Yaskawa INFORM job: A_ROOF_UPPER_0614_2_PAINT_2.JBI

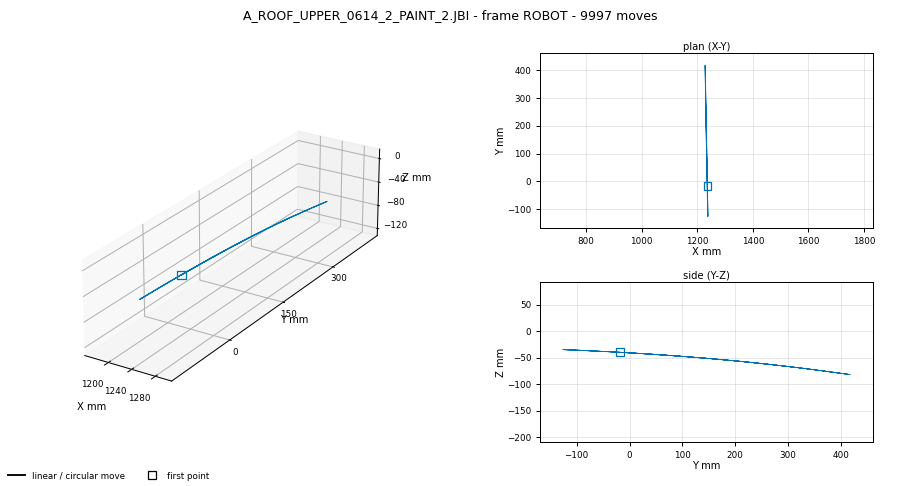
[picture p0: tool path of A_ROOF_UPPER_0614_2_PAINT_2.JBI in frame ROBOT, 9997 of 9997 moves have a stored position in this frame; points joined in program order, loops and branches not executed]
/JOB
//NAME A_ROOF_UPPER_0614_2_PAINT2
//POS
///NPOS 9997,0,0,0,0,0
///TOOL 1
///USER 0
///POSTYPE ROBOT
///RECTAN
///RCONF 1,0,0,0,0,0,0,0,0,0,0,0,0,0,0,0,0,0,0,0,0,0,0,0
C00000=1236.915,-17.452,-39.644,-179.558,5.242,148.773
C00001=1236.910,-17.203,-39.658,-179.555,5.243,148.772
C00002=1236.905,-16.953,-39.672,-179.553,5.243,148.771
C00003=1236.900,-16.704,-39.686,-179.551,5.243,148.771
C00004=1236.895,-16.454,-39.700,-179.548,5.244,148.770
C00005=1236.890,-16.204,-39.714,-179.546,5.243,148.769
C00006=1236.884,-15.955,-39.728,-179.543,5.244,148.769
C00007=1236.880,-15.705,-39.741,-179.541,5.244,148.768
C00008=1236.875,-15.456,-39.756,-179.539,5.244,148.767
C00009=1236.870,-15.206,-39.770,-179.536,5.245,148.767
C00010=1236.864,-14.956,-39.783,-179.534,5.244,148.766
C00011=1236.859,-14.707,-39.798,-179.531,5.245,148.765
C00012=1236.854,-14.457,-39.812,-179.528,5.245,148.764
C00013=1236.849,-14.207,-39.826,-179.526,5.245,148.764
C00014=1236.844,-13.959,-39.839,-179.523,5.245,148.763
C00015=1236.839,-13.709,-39.854,-179.521,5.246,148.762
C00016=1236.834,-13.459,-39.868,-179.519,5.246,148.761
C00017=1236.829,-13.209,-39.882,-179.516,5.246,148.761
C00018=1236.824,-12.960,-39.896,-179.513,5.247,148.760
C00019=1236.819,-12.711,-39.910,-179.511,5.246,148.759
C00020=1236.814,-12.461,-39.925,-179.508,5.247,148.759
C00021=1236.809,-12.211,-39.938,-179.506,5.247,148.758
C00022=1236.803,-11.962,-39.952,-179.504,5.247,148.757
C00023=1236.799,-11.712,-39.966,-179.501,5.248,148.757
C00024=1236.794,-11.463,-39.980,-179.499,5.247,148.756
C00025=1236.789,-11.213,-39.994,-179.496,5.248,148.755
C00026=1236.784,-10.964,-40.008,-179.494,5.248,148.755
C00027=1236.779,-10.714,-40.023,-179.492,5.248,148.754
C00028=1236.774,-10.464,-40.037,-179.488,5.248,148.753
C00029=1236.769,-10.215,-40.051,-179.486,5.249,148.752
C00030=1236.764,-9.965,-40.065,-179.484,5.249,148.752
C00031=1236.758,-9.716,-40.079,-179.481,5.249,148.751
C00032=1236.753,-9.466,-40.094,-179.478,5.250,148.750
C00033=1236.748,-9.217,-40.108,-179.476,5.249,148.749
C00034=1236.743,-8.967,-40.122,-179.474,5.250,148.749
C00035=1236.739,-8.718,-40.137,-179.471,5.250,148.748
C00036=1236.734,-8.468,-40.151,-179.469,5.250,148.747
C00037=1236.728,-8.219,-40.165,-179.466,5.251,148.747
C00038=1236.723,-7.969,-40.180,-179.464,5.251,148.746
C00039=1236.718,-7.720,-40.194,-179.462,5.251,148.745
C00040=1236.713,-7.470,-40.208,-179.459,5.251,148.745
C00041=1236.708,-7.220,-40.222,-179.456,5.252,148.744
C00042=1236.703,-6.970,-40.237,-179.454,5.252,148.743
C00043=1236.698,-6.721,-40.251,-179.451,5.252,148.743
C00044=1236.693,-6.472,-40.265,-179.448,5.252,148.742
C00045=1236.688,-6.223,-40.280,-179.446,5.252,148.741
C00046=1236.683,-5.973,-40.294,-179.444,5.253,148.740
C00047=1236.678,-5.723,-40.308,-179.441,5.253,148.740
C00048=1236.673,-5.474,-40.323,-179.439,5.253,148.739
C00049=1236.668,-5.224,-40.337,-179.436,5.253,148.738
C00050=1236.663,-4.975,-40.351,-179.434,5.254,148.737
C00051=1236.658,-4.725,-40.365,-179.431,5.254,148.737
C00052=1236.653,-4.476,-40.380,-179.429,5.254,148.736
C00053=1236.648,-4.226,-40.394,-179.426,5.255,148.735
C00054=1236.643,-3.976,-40.409,-179.424,5.254,148.735
C00055=1236.638,-3.727,-40.424,-179.421,5.255,148.734
C00056=1236.633,-3.477,-40.438,-179.419,5.255,148.733
C00057=1236.628,-3.228,-40.453,-179.417,5.255,148.733
C00058=1236.623,-2.978,-40.467,-179.414,5.256,148.732
C00059=1236.617,-2.729,-40.481,-179.411,5.256,148.731
C00060=1236.613,-2.479,-40.495,-179.409,5.256,148.731
C00061=1236.608,-2.230,-40.510,-179.407,5.256,148.730
C00062=1236.603,-1.981,-40.525,-179.404,5.257,148.729
C00063=1236.597,-1.731,-40.540,-179.401,5.256,148.728
C00064=1236.592,-1.481,-40.554,-179.399,5.257,148.728
C00065=1236.588,-1.232,-40.569,-179.396,5.257,148.727
C00066=1236.583,-0.982,-40.583,-179.394,5.257,148.726
C00067=1236.578,-0.732,-40.597,-179.391,5.258,148.725
C00068=1236.573,-0.483,-40.612,-179.389,5.258,148.725
C00069=1236.568,-0.233,-40.627,-179.387,5.258,148.724
C00070=1236.562,0.017,-40.641,-179.384,5.258,148.723
C00071=1236.558,0.266,-40.656,-179.381,5.259,148.723
C00072=1236.552,0.515,-40.670,-179.379,5.259,148.722
C00073=1236.547,0.764,-40.685,-179.377,5.259,148.721
C00074=1236.543,1.013,-40.700,-179.374,5.260,148.721
C00075=1236.537,1.263,-40.715,-179.371,5.260,148.720
C00076=1236.532,1.513,-40.729,-179.369,5.260,148.719
C00077=1236.527,1.762,-40.744,-179.367,5.261,148.719
C00078=1236.522,2.012,-40.758,-179.364,5.261,148.718
C00079=1236.518,2.261,-40.773,-179.362,5.261,148.717
C00080=1236.512,2.511,-40.788,-179.359,5.261,148.717
C00081=1236.507,2.761,-40.802,-179.357,5.262,148.716
C00082=1236.502,3.010,-40.817,-179.354,5.262,148.715
C00083=1236.497,3.260,-40.831,-179.352,5.262,148.714
C00084=1236.492,3.529,-40.848,-179.349,5.262,148.714
C00085=1236.486,3.797,-40.863,-179.346,5.263,148.713
C00086=1236.481,4.066,-40.879,-179.343,5.263,148.712
C00087=1236.475,4.335,-40.895,-179.341,5.263,148.711
C00088=1236.471,4.584,-40.910,-179.338,5.263,148.711
C00089=1236.466,4.834,-40.925,-179.335,5.264,148.710
C00090=1236.461,5.083,-40.940,-179.333,5.264,148.709
C00091=1236.456,5.333,-40.955,-179.331,5.264,148.709
C00092=1236.451,5.582,-40.970,-179.328,5.265,148.708
C00093=1236.446,5.832,-40.984,-179.325,5.265,148.707
C00094=1236.441,6.082,-40.999,-179.323,5.265,148.706
C00095=1236.436,6.331,-41.014,-179.321,5.265,148.706
C00096=1236.431,6.580,-41.029,-179.318,5.266,148.705
C00097=1236.425,6.830,-41.044,-179.315,5.266,148.704
C00098=1236.421,7.079,-41.059,-179.313,5.266,148.704
C00099=1236.416,7.329,-41.073,-179.311,5.267,148.703
C00100=1236.410,7.579,-41.088,-179.308,5.267,148.702
C00101=1236.405,7.828,-41.103,-179.306,5.267,148.702
C00102=1236.401,8.077,-41.118,-179.303,5.268,148.701
C00103=1236.395,8.327,-41.133,-179.301,5.268,148.700
C00104=1236.391,8.577,-41.148,-179.298,5.269,148.700
C00105=1236.386,8.826,-41.163,-179.296,5.268,148.699
C00106=1236.381,9.076,-41.178,-179.293,5.269,148.698
C00107=1236.376,9.325,-41.193,-179.291,5.269,148.698
C00108=1236.371,9.575,-41.207,-179.289,5.269,148.697
C00109=1236.366,9.824,-41.223,-179.286,5.270,148.696
C00110=1236.361,10.074,-41.238,-179.283,5.270,148.695
C00111=1236.355,10.324,-41.253,-179.281,5.271,148.695
C00112=1236.351,10.573,-41.268,-179.279,5.271,148.694
C00113=1236.346,10.822,-41.283,-179.276,5.271,148.693
C00114=1236.340,11.072,-41.297,-179.273,5.272,148.693
C00115=1236.336,11.321,-41.312,-179.271,5.271,148.692
C00116=1236.331,11.571,-41.328,-179.268,5.272,148.691
C00117=1236.326,11.821,-41.343,-179.265,5.272,148.690
C00118=1236.320,12.070,-41.358,-179.263,5.273,148.690
C00119=1236.316,12.319,-41.373,-179.261,5.272,148.689
C00120=1236.311,12.569,-41.388,-179.258,5.273,148.688
C00121=1236.305,12.818,-41.403,-179.255,5.273,148.688
C00122=1236.301,13.067,-41.418,-179.253,5.274,148.687
C00123=1236.295,13.317,-41.434,-179.251,5.274,148.686
C00124=1236.291,13.567,-41.448,-179.248,5.274,148.686
C00125=1236.286,13.817,-41.464,-179.245,5.275,148.685
C00126=1236.281,14.066,-41.479,-179.243,5.275,148.684
C00127=1236.276,14.315,-41.494,-179.241,5.275,148.684
C00128=1236.271,14.565,-41.509,-179.238,5.276,148.683
C00129=1236.265,14.814,-41.524,-179.235,5.276,148.682
C00130=1236.261,15.063,-41.539,-179.233,5.276,148.682
C00131=1236.256,15.313,-41.555,-179.231,5.276,148.681
C00132=1236.251,15.562,-41.570,-179.228,5.277,148.680
C00133=1236.246,15.813,-41.585,-179.225,5.278,148.679
C00134=1236.241,16.062,-41.600,-179.223,5.277,148.679
C00135=1236.236,16.311,-41.616,-179.221,5.278,148.678
C00136=1236.231,16.560,-41.631,-179.218,5.278,148.677
C00137=1236.226,16.810,-41.647,-179.215,5.279,148.677
C00138=1236.221,17.059,-41.662,-179.213,5.279,148.676
C00139=1236.216,17.309,-41.677,-179.211,5.279,148.675
C00140=1236.210,17.559,-41.692,-179.208,5.280,148.675
C00141=1236.206,17.808,-41.707,-179.205,5.280,148.674
C00142=1236.201,18.058,-41.723,-179.203,5.280,148.673
C00143=1236.196,18.307,-41.738,-179.201,5.281,148.673
C00144=1236.191,18.556,-41.754,-179.198,5.281,148.672
C00145=1236.186,18.805,-41.769,-179.195,5.282,148.671
C00146=1236.181,19.055,-41.784,-179.193,5.281,148.671
C00147=1236.176,19.305,-41.800,-179.190,5.282,148.670
C00148=1236.171,19.554,-41.815,-179.188,5.283,148.669
C00149=1236.166,19.804,-41.830,-179.185,5.283,148.669
C00150=1236.161,20.053,-41.845,-179.183,5.283,148.668
C00151=1236.156,20.303,-41.861,-179.180,5.283,148.667
C00152=1236.151,20.553,-41.877,-179.178,5.284,148.666
C00153=1236.146,20.802,-41.892,-179.175,5.284,148.666
C00154=1236.141,21.051,-41.907,-179.173,5.284,148.665
C00155=1236.135,21.301,-41.923,-179.170,5.285,148.664
C00156=1236.131,21.550,-41.938,-179.168,5.285,148.664
C00157=1236.126,21.800,-41.954,-179.165,5.286,148.663
C00158=1236.121,22.049,-41.969,-179.163,5.286,148.662
C00159=1236.116,22.298,-41.984,-179.160,5.286,148.662
C00160=1236.111,22.548,-42.000,-179.158,5.287,148.661
C00161=1236.107,22.797,-42.015,-179.155,5.287,148.660
C00162=1236.101,23.047,-42.031,-179.153,5.288,148.660
C00163=1236.096,23.297,-42.047,-179.150,5.288,148.659
C00164=1236.091,23.546,-42.062,-179.148,5.288,148.658
C00165=1236.086,23.795,-42.077,-179.145,5.289,148.658
C00166=1236.081,24.044,-42.094,-179.143,5.289,148.657
C00167=1236.076,24.294,-42.110,-179.140,5.289,148.656
C00168=1236.072,24.543,-42.125,-179.138,5.290,148.656
C00169=1236.066,24.793,-42.140,-179.135,5.290,148.655
C00170=1236.062,25.043,-42.156,-179.132,5.291,148.654
C00171=1236.057,25.292,-42.171,-179.130,5.291,148.654
C00172=1236.052,25.541,-42.187,-179.128,5.291,148.653
C00173=1236.047,25.792,-42.203,-179.125,5.291,148.652
C00174=1236.041,26.041,-42.218,-179.122,5.292,148.652
C00175=1236.037,26.289,-42.234,-179.120,5.293,148.651
C00176=1236.032,26.539,-42.250,-179.118,5.292,148.650
C00177=1236.027,26.789,-42.266,-179.115,5.293,148.649
C00178=1236.022,27.038,-42.281,-179.112,5.293,148.649
C00179=1236.017,27.287,-42.296,-179.110,5.294,148.648
C00180=1236.012,27.538,-42.312,-179.107,5.295,148.647
C00181=1236.007,27.786,-42.328,-179.105,5.294,148.647
C00182=1236.002,28.036,-42.344,-179.102,5.295,148.646
C00183=1235.997,28.286,-42.360,-179.100,5.295,148.645
C00184=1235.992,28.535,-42.375,-179.097,5.296,148.645
C00185=1235.987,28.785,-42.391,-179.095,5.296,148.644
C00186=1235.982,29.034,-42.407,-179.092,5.296,148.643
C00187=1235.977,29.283,-42.423,-179.090,5.297,148.643
C00188=1235.971,29.552,-42.440,-179.087,5.297,148.642
C00189=1235.966,29.821,-42.457,-179.085,5.298,148.641
C00190=1235.961,30.089,-42.474,-179.081,5.298,148.640
C00191=1235.956,30.358,-42.491,-179.079,5.299,148.640
C00192=1235.951,30.607,-42.506,-179.076,5.299,148.639
C00193=1235.946,30.857,-42.522,-179.074,5.299,148.638
C00194=1235.941,31.106,-42.538,-179.071,5.300,148.638
C00195=1235.936,31.356,-42.554,-179.069,5.300,148.637
C00196=1235.931,31.605,-42.570,-179.066,5.301,148.636
C00197=1235.926,31.854,-42.586,-179.063,5.301,148.636
C00198=1235.922,32.104,-42.602,-179.061,5.301,148.635
C00199=1235.916,32.353,-42.617,-179.059,5.302,148.634
C00200=1235.912,32.603,-42.634,-179.056,5.302,148.634
C00201=1235.906,32.852,-42.649,-179.053,5.303,148.633
C00202=1235.901,33.102,-42.665,-179.051,5.303,148.632
C00203=1235.896,33.351,-42.682,-179.049,5.303,148.632
C00204=1235.891,33.600,-42.697,-179.046,5.304,148.631
C00205=1235.886,33.851,-42.713,-179.043,5.304,148.630
C00206=1235.881,34.099,-42.730,-179.041,5.305,148.630
C00207=1235.876,34.349,-42.746,-179.038,5.305,148.629
C00208=1235.871,34.598,-42.762,-179.037,5.305,148.628
C00209=1235.867,34.847,-42.777,-179.034,5.306,148.628
C00210=1235.862,35.097,-42.794,-179.031,5.307,148.627
C00211=1235.857,35.346,-42.809,-179.029,5.307,148.626
C00212=1235.852,35.596,-42.825,-179.026,5.308,148.626
C00213=1235.847,35.845,-42.841,-179.023,5.308,148.625
C00214=1235.842,36.095,-42.857,-179.021,5.308,148.624
C00215=1235.837,36.344,-42.874,-179.019,5.309,148.624
C00216=1235.832,36.594,-42.890,-179.016,5.309,148.623
C00217=1235.827,36.843,-42.906,-179.013,5.310,148.622
C00218=1235.822,37.093,-42.922,-179.011,5.310,148.622
C00219=1235.817,37.342,-42.938,-179.009,5.310,148.621
C00220=1235.813,37.592,-42.954,-179.006,5.311,148.620
C00221=1235.807,37.841,-42.970,-179.003,5.311,148.620
C00222=1235.803,38.091,-42.986,-179.001,5.312,148.619
C00223=1235.798,38.340,-43.003,-178.998,5.312,148.618
C00224=1235.793,38.590,-43.019,-178.995,5.313,148.618
C00225=1235.788,38.838,-43.035,-178.993,5.313,148.617
C00226=1235.783,39.089,-43.051,-178.991,5.313,148.616
C00227=1235.778,39.337,-43.067,-178.988,5.314,148.616
C00228=1235.773,39.587,-43.084,-178.985,5.314,148.615
C00229=1235.767,39.837,-43.100,-178.983,5.315,148.614
C00230=1235.763,40.086,-43.117,-178.980,5.315,148.614
C00231=1235.757,40.335,-43.132,-178.978,5.315,148.613
C00232=1235.753,40.585,-43.149,-178.975,5.316,148.612
C00233=1235.747,40.834,-43.165,-178.973,5.316,148.612
C00234=1235.743,41.084,-43.181,-178.971,5.317,148.611
C00235=1235.738,41.333,-43.197,-178.968,5.318,148.610
C00236=1235.733,41.583,-43.213,-178.965,5.318,148.610
C00237=1235.728,41.831,-43.230,-178.963,5.318,148.609
C00238=1235.724,42.081,-43.246,-178.961,5.319,148.608
C00239=1235.718,42.330,-43.262,-178.958,5.319,148.608
C00240=1235.713,42.580,-43.279,-178.955,5.320,148.607
C00241=1235.708,42.829,-43.296,-178.953,5.320,148.606
C00242=1235.703,43.079,-43.312,-178.950,5.321,148.606
C00243=1235.699,43.329,-43.328,-178.948,5.322,148.605
C00244=1235.694,43.577,-43.345,-178.945,5.321,148.604
C00245=1235.689,43.827,-43.360,-178.943,5.322,148.604
C00246=1235.684,44.076,-43.377,-178.940,5.322,148.603
C00247=1235.678,44.326,-43.394,-178.938,5.323,148.602
C00248=1235.674,44.575,-43.411,-178.935,5.324,148.602
C00249=1235.669,44.825,-43.426,-178.932,5.324,148.601
C00250=1235.664,45.074,-43.443,-178.930,5.325,148.600
C00251=1235.659,45.323,-43.459,-178.928,5.324,148.600
C00252=1235.655,45.573,-43.476,-178.925,5.325,148.599
C00253=1235.648,45.822,-43.492,-178.923,5.326,148.599
C00254=1235.644,46.072,-43.509,-178.920,5.327,148.598
C00255=1235.639,46.321,-43.525,-178.917,5.327,148.597
C00256=1235.634,46.570,-43.542,-178.915,5.328,148.596
C00257=1235.630,46.820,-43.558,-178.912,5.328,148.596
C00258=1235.624,47.070,-43.575,-178.910,5.328,148.595
C00259=1235.619,47.319,-43.591,-178.908,5.329,148.594
C00260=1235.615,47.568,-43.608,-178.905,5.329,148.594
C00261=1235.610,47.817,-43.624,-178.902,5.330,148.593
C00262=1235.605,48.067,-43.642,-178.900,5.330,148.592
C00263=1235.600,48.317,-43.657,-178.897,5.331,148.592
C00264=1235.595,48.566,-43.674,-178.894,5.331,148.591
C00265=1235.590,48.815,-43.690,-178.892,5.331,148.590
C00266=1235.585,49.065,-43.708,-178.890,5.332,148.590
C00267=1235.580,49.314,-43.724,-178.887,5.333,148.589
C00268=1235.575,49.563,-43.741,-178.885,5.333,148.589
C00269=1235.571,49.813,-43.757,-178.882,5.334,148.588
C00270=1235.565,50.062,-43.774,-178.880,5.334,148.587
C00271=1235.561,50.311,-43.791,-178.877,5.335,148.587
C00272=1235.556,50.561,-43.808,-178.874,5.336,148.586
C00273=1235.550,50.811,-43.824,-178.872,5.335,148.585
C00274=1235.546,51.060,-43.840,-178.870,5.336,148.585
C00275=1235.541,51.309,-43.857,-178.867,5.337,148.584
C00276=1235.535,51.559,-43.874,-178.864,5.337,148.583
C00277=1235.531,51.808,-43.891,-178.862,5.338,148.583
C00278=1235.526,52.058,-43.907,-178.859,5.338,148.582
C00279=1235.521,52.307,-43.925,-178.857,5.339,148.582
C00280=1235.516,52.556,-43.941,-178.854,5.340,148.581
C00281=1235.511,52.806,-43.958,-178.852,5.340,148.580
C00282=1235.506,53.055,-43.975,-178.850,5.340,148.580
C00283=1235.501,53.304,-43.991,-178.847,5.341,148.579
C00284=1235.497,53.554,-44.008,-178.844,5.341,148.578
C00285=1235.491,53.803,-44.025,-178.842,5.342,148.577
C00286=1235.487,54.053,-44.042,-178.839,5.342,148.577
C00287=1235.482,54.302,-44.058,-178.836,5.343,148.576
C00288=1235.477,54.552,-44.075,-178.834,5.344,148.575
C00289=1235.473,54.800,-44.093,-178.831,5.344,148.575
C00290=1235.467,55.049,-44.110,-178.829,5.345,148.574
C00291=1235.462,55.299,-44.126,-178.826,5.346,148.574
C00292=1235.457,55.568,-44.145,-178.823,5.346,148.573
C00293=1235.452,55.836,-44.163,-178.821,5.347,148.572
C00294=1235.446,56.105,-44.181,-178.818,5.347,148.571
C00295=1235.441,56.372,-44.199,-178.815,5.348,148.571
C00296=1235.436,56.622,-44.216,-178.813,5.348,148.570
C00297=1235.431,56.872,-44.233,-178.810,5.349,148.569
C00298=1235.427,57.121,-44.250,-178.808,5.349,148.569
C00299=1235.422,57.371,-44.267,-178.806,5.350,148.568
C00300=1235.416,57.620,-44.283,-178.803,5.350,148.568
C00301=1235.411,57.870,-44.301,-178.801,5.351,148.567
C00302=1235.407,58.118,-44.318,-178.798,5.351,148.566
C00303=1235.402,58.368,-44.335,-178.795,5.352,148.566
C00304=1235.397,58.617,-44.352,-178.793,5.352,148.565
C00305=1235.392,58.867,-44.369,-178.790,5.353,148.564
C00306=1235.387,59.116,-44.385,-178.787,5.354,148.564
C00307=1235.382,59.365,-44.403,-178.785,5.354,148.563
C00308=1235.378,59.615,-44.420,-178.782,5.355,148.562
C00309=1235.372,59.864,-44.437,-178.781,5.355,148.562
C00310=1235.367,60.114,-44.454,-178.778,5.356,148.561
C00311=1235.362,60.363,-44.472,-178.775,5.356,148.561
C00312=1235.358,60.612,-44.488,-178.773,5.357,148.560
C00313=1235.353,60.862,-44.506,-178.770,5.357,148.559
C00314=1235.348,61.111,-44.522,-178.767,5.358,148.559
C00315=1235.343,61.360,-44.540,-178.765,5.358,148.558
C00316=1235.338,61.610,-44.557,-178.762,5.359,148.557
C00317=1235.333,61.859,-44.574,-178.759,5.360,148.557
C00318=1235.328,62.108,-44.592,-178.757,5.361,148.556
C00319=1235.324,62.358,-44.608,-178.755,5.361,148.556
C00320=1235.318,62.608,-44.626,-178.752,5.362,148.555
C00321=1235.314,62.857,-44.642,-178.749,5.362,148.554
C00322=1235.309,63.106,-44.660,-178.747,5.363,148.554
C00323=1235.303,63.355,-44.677,-178.745,5.363,148.553
C00324=1235.299,63.604,-44.695,-178.742,5.363,148.552
C00325=1235.294,63.854,-44.712,-178.739,5.364,148.552
C00326=1235.289,64.104,-44.729,-178.737,5.365,148.551
C00327=1235.285,64.353,-44.747,-178.735,5.365,148.550
C00328=1235.279,64.603,-44.764,-178.732,5.366,148.550
C00329=1235.275,64.852,-44.780,-178.729,5.367,148.549
C00330=1235.269,65.100,-44.798,-178.727,5.367,148.548
C00331=1235.264,65.350,-44.815,-178.724,5.368,148.548
C00332=1235.260,65.599,-44.833,-178.722,5.368,148.547
C00333=1235.255,65.849,-44.850,-178.719,5.369,148.547
C00334=1235.251,66.098,-44.867,-178.717,5.370,148.546
C00335=1235.245,66.348,-44.885,-178.714,5.370,148.545
C00336=1235.240,66.597,-44.903,-178.712,5.371,148.545
C00337=1235.236,66.846,-44.919,-178.709,5.372,148.544
C00338=1235.231,67.096,-44.937,-178.706,5.372,148.543
C00339=1235.226,67.345,-44.955,-178.704,5.373,148.543
C00340=1235.221,67.595,-44.972,-178.701,5.373,148.542
C00341=1235.216,67.843,-44.989,-178.699,5.374,148.542
C00342=1235.211,68.093,-45.006,-178.697,5.374,148.541
C00343=1235.206,68.342,-45.024,-178.694,5.375,148.540
C00344=1235.201,68.592,-45.041,-178.692,5.375,148.540
C00345=1235.196,68.841,-45.059,-178.689,5.376,148.539
C00346=1235.191,69.090,-45.077,-178.686,5.377,148.538
C00347=1235.186,69.340,-45.094,-178.684,5.377,148.538
C00348=1235.182,69.589,-45.111,-178.682,5.378,148.537
C00349=1235.177,69.838,-45.129,-178.679,5.379,148.537
C00350=1235.172,70.088,-45.147,-178.676,5.379,148.536
C00351=1235.167,70.337,-45.164,-178.674,5.380,148.535
C00352=1235.162,70.586,-45.181,-178.671,5.380,148.535
C00353=1235.158,70.835,-45.199,-178.668,5.381,148.534
C00354=1235.152,71.085,-45.216,-178.666,5.382,148.533
C00355=1235.147,71.334,-45.234,-178.664,5.383,148.533
C00356=1235.143,71.584,-45.251,-178.661,5.383,148.532
C00357=1235.138,71.833,-45.269,-178.658,5.384,148.531
C00358=1235.133,72.082,-45.287,-178.656,5.384,148.531
C00359=1235.128,72.332,-45.304,-178.653,5.385,148.530
C00360=1235.123,72.581,-45.322,-178.650,5.386,148.529
C00361=1235.119,72.830,-45.340,-178.648,5.386,148.529
C00362=1235.114,73.080,-45.357,-178.646,5.387,148.528
C00363=1235.109,73.329,-45.375,-178.643,5.388,148.528
C00364=1235.104,73.578,-45.393,-178.640,5.388,148.527
C00365=1235.099,73.827,-45.411,-178.638,5.389,148.526
C00366=1235.094,74.077,-45.428,-178.635,5.389,148.526
C00367=1235.089,74.326,-45.446,-178.633,5.390,148.525
C00368=1235.085,74.575,-45.464,-178.630,5.391,148.525
C00369=1235.079,74.825,-45.481,-178.628,5.392,148.524
C00370=1235.074,75.074,-45.499,-178.625,5.392,148.523
C00371=1235.069,75.323,-45.517,-178.623,5.393,148.523
C00372=1235.065,75.573,-45.535,-178.620,5.393,148.522
C00373=1235.059,75.822,-45.552,-178.618,5.394,148.522
C00374=1235.054,76.072,-45.570,-178.615,5.395,148.521
C00375=1235.050,76.321,-45.588,-178.613,5.396,148.520
C00376=1235.046,76.570,-45.606,-178.610,5.396,148.520
C00377=1235.041,76.819,-45.624,-178.607,5.397,148.519
C00378=1235.036,77.069,-45.641,-178.605,5.398,148.519
C00379=1235.031,77.318,-45.659,-178.603,5.398,148.518
C00380=1235.026,77.568,-45.677,-178.600,5.399,148.517
C00381=1235.021,77.817,-45.695,-178.597,5.400,148.517
C00382=1235.016,78.066,-45.713,-178.595,5.400,148.516
C00383=1235.011,78.315,-45.731,-178.592,5.401,148.515
C00384=1235.006,78.564,-45.749,-178.590,5.402,148.515
C00385=1235.001,78.814,-45.766,-178.587,5.402,148.514
C00386=1234.996,79.063,-45.784,-178.585,5.403,148.513
C00387=1234.992,79.313,-45.802,-178.582,5.403,148.513
C00388=1234.987,79.562,-45.820,-178.579,5.404,148.512
C00389=1234.982,79.812,-45.838,-178.577,5.405,148.512
C00390=1234.977,80.061,-45.856,-178.575,5.406,148.511
C00391=1234.972,80.310,-45.874,-178.572,5.406,148.510
C00392=1234.967,80.559,-45.892,-178.569,5.407,148.510
C00393=1234.962,80.808,-45.910,-178.567,5.407,148.509
C00394=1234.958,81.057,-45.928,-178.565,5.408,148.509
C00395=1234.953,81.307,-45.946,-178.562,5.409,148.508
C00396=1234.948,81.576,-45.965,-178.559,5.410,148.507
C00397=1234.943,81.844,-45.985,-178.557,5.410,148.507
C00398=1234.938,82.113,-46.004,-178.554,5.411,148.506
C00399=1234.933,82.381,-46.024,-178.551,5.412,148.505
C00400=1234.927,82.630,-46.042,-178.548,5.413,148.505
C00401=1234.922,82.880,-46.060,-178.546,5.413,148.504
C00402=1234.917,83.129,-46.078,-178.543,5.414,148.503
C00403=1234.912,83.378,-46.096,-178.540,5.415,148.503
C00404=1234.907,83.627,-46.114,-178.538,5.416,148.502
C00405=1234.903,83.877,-46.132,-178.536,5.416,148.502
C00406=1234.898,84.126,-46.150,-178.533,5.417,148.501
C00407=1234.893,84.375,-46.168,-178.530,5.417,148.500
C00408=1234.889,84.624,-46.187,-178.528,5.418,148.500
C00409=1234.884,84.873,-46.205,-178.526,5.419,148.499
C00410=1234.879,85.122,-46.223,-178.523,5.420,148.499
C00411=1234.874,85.372,-46.241,-178.520,5.420,148.498
C00412=1234.869,85.622,-46.260,-178.518,5.421,148.497
C00413=1234.864,85.871,-46.278,-178.516,5.422,148.497
C00414=1234.859,86.120,-46.296,-178.513,5.422,148.496
C00415=1234.855,86.370,-46.314,-178.510,5.423,148.496
C00416=1234.850,86.619,-46.332,-178.508,5.424,148.495
C00417=1234.845,86.868,-46.351,-178.505,5.424,148.494
C00418=1234.840,87.117,-46.369,-178.503,5.425,148.494
C00419=1234.835,87.366,-46.387,-178.500,5.426,148.493
C00420=1234.830,87.616,-46.406,-178.498,5.426,148.493
C00421=1234.825,87.865,-46.424,-178.495,5.427,148.492
C00422=1234.820,88.114,-46.442,-178.493,5.429,148.492
C00423=1234.816,88.363,-46.460,-178.490,5.429,148.491
C00424=1234.811,88.613,-46.479,-178.487,5.430,148.490
C00425=1234.806,88.862,-46.497,-178.485,5.431,148.490
C00426=1234.801,89.112,-46.515,-178.483,5.432,148.489
C00427=1234.796,89.360,-46.534,-178.480,5.432,148.488
C00428=1234.792,89.610,-46.552,-178.477,5.433,148.488
C00429=1234.786,89.859,-46.571,-178.475,5.433,148.487
C00430=1234.781,90.109,-46.589,-178.472,5.434,148.487
C00431=1234.777,90.357,-46.608,-178.470,5.435,148.486
C00432=1234.773,90.607,-46.626,-178.467,5.436,148.485
C00433=1234.767,90.857,-46.645,-178.465,5.436,148.485
C00434=1234.762,91.106,-46.663,-178.462,5.437,148.484
C00435=1234.758,91.355,-46.682,-178.460,5.438,148.484
C00436=1234.753,91.604,-46.700,-178.457,5.438,148.483
C00437=1234.747,91.854,-46.718,-178.455,5.439,148.482
C00438=1234.743,92.103,-46.737,-178.451,5.440,148.482
C00439=1234.738,92.352,-46.755,-178.449,5.441,148.481
C00440=1234.734,92.601,-46.773,-178.447,5.442,148.481
C00441=1234.728,92.850,-46.793,-178.444,5.443,148.480
C00442=1234.724,93.100,-46.811,-178.441,5.443,148.479
C00443=1234.719,93.349,-46.830,-178.439,5.444,148.479
C00444=1234.714,93.598,-46.848,-178.437,5.445,148.478
C00445=1234.709,93.848,-46.866,-178.434,5.445,148.478
C00446=1234.705,94.096,-46.885,-178.432,5.446,148.477
C00447=1234.699,94.346,-46.904,-178.429,5.447,148.477
C00448=1234.695,94.595,-46.923,-178.427,5.448,148.476
C00449=1234.690,94.844,-46.941,-178.424,5.448,148.475
C00450=1234.685,95.094,-46.959,-178.421,5.450,148.475
C00451=1234.681,95.343,-46.978,-178.419,5.451,148.474
C00452=1234.676,95.592,-46.996,-178.416,5.451,148.474
C00453=1234.671,95.842,-47.016,-178.414,5.452,148.473
C00454=1234.666,96.091,-47.034,-178.411,5.452,148.472
C00455=1234.661,96.340,-47.053,-178.409,5.453,148.472
C00456=1234.656,96.590,-47.072,-178.406,5.454,148.471
C00457=1234.652,96.838,-47.090,-178.404,5.455,148.471
C00458=1234.646,97.088,-47.109,-178.401,5.455,148.470
C00459=1234.642,97.337,-47.128,-178.399,5.456,148.470
C00460=1234.636,97.587,-47.147,-178.396,5.457,148.469
C00461=1234.632,97.836,-47.166,-178.393,5.458,148.468
C00462=1234.627,98.085,-47.184,-178.391,5.459,148.468
C00463=1234.622,98.334,-47.203,-178.388,5.460,148.467
C00464=1234.618,98.583,-47.222,-178.386,5.460,148.467
C00465=1234.612,98.833,-47.241,-178.383,5.461,148.466
C00466=1234.608,99.082,-47.260,-178.381,5.462,148.465
C00467=1234.603,99.331,-47.278,-178.378,5.463,148.465
C00468=1234.598,99.580,-47.297,-178.376,5.463,148.464
C00469=1234.593,99.830,-47.316,-178.374,5.464,148.464
C00470=1234.589,100.079,-47.335,-178.370,5.466,148.463
C00471=1234.584,100.328,-47.354,-178.368,5.466,148.462
C00472=1234.579,100.577,-47.372,-178.365,5.467,148.462
C00473=1234.574,100.827,-47.392,-178.363,5.468,148.461
C00474=1234.570,101.076,-47.410,-178.360,5.469,148.461
C00475=1234.564,101.325,-47.429,-178.358,5.469,148.460
C00476=1234.560,101.574,-47.448,-178.356,5.470,148.460
C00477=1234.555,101.823,-47.467,-178.353,5.471,148.459
C00478=1234.550,102.073,-47.486,-178.350,5.472,148.458
C00479=1234.545,102.322,-47.505,-178.347,5.473,148.458
C00480=1234.541,102.571,-47.524,-178.345,5.474,148.457
C00481=1234.535,102.821,-47.543,-178.343,5.474,148.457
C00482=1234.531,103.070,-47.562,-178.340,5.475,148.456
C00483=1234.526,103.319,-47.581,-178.338,5.476,148.456
C00484=1234.522,103.568,-47.600,-178.335,5.477,148.455
C00485=1234.516,103.818,-47.619,-178.333,5.477,148.454
C00486=1234.512,104.067,-47.638,-178.329,5.479,148.454
C00487=1234.507,104.316,-47.657,-178.327,5.480,148.453
C00488=1234.502,104.565,-47.677,-178.325,5.480,148.453
C00489=1234.497,104.814,-47.695,-178.322,5.481,148.452
C00490=1234.492,105.064,-47.714,-178.320,5.482,148.452
C00491=1234.488,105.313,-47.733,-178.317,5.482,148.451
C00492=1234.483,105.562,-47.753,-178.315,5.483,148.450
C00493=1234.478,105.811,-47.772,-178.312,5.485,148.450
C00494=1234.474,106.060,-47.791,-178.309,5.486,148.449
C00495=1234.468,106.310,-47.810,-178.307,5.486,148.449
C00496=1234.463,106.559,-47.829,-178.305,5.487,148.448
C00497=1234.459,106.808,-47.848,-178.302,5.488,148.448
C00498=1234.454,107.057,-47.868,-178.299,5.488,148.447
C00499=1234.449,107.306,-47.886,-178.297,5.489,148.446
C00500=1234.445,107.575,-47.907,-178.294,5.491,148.446
C00501=1234.439,107.844,-47.928,-178.292,5.491,148.445
C00502=1234.434,108.112,-47.948,-178.289,5.492,148.445
C00503=1234.429,108.380,-47.970,-178.286,5.493,148.444
C00504=1234.424,108.629,-47.989,-178.283,5.494,148.443
C00505=1234.420,108.879,-48.008,-178.281,5.495,148.443
C00506=1234.414,109.127,-48.027,-178.278,5.496,148.442
C00507=1234.409,109.377,-48.047,-178.276,5.496,148.442
C00508=1234.405,109.627,-48.067,-178.273,5.498,148.441
C00509=1234.400,109.875,-48.085,-178.270,5.499,148.441
C00510=1234.395,110.125,-48.105,-178.268,5.499,148.440
C00511=1234.390,110.374,-48.123,-178.266,5.500,148.439
C00512=1234.386,110.623,-48.143,-178.263,5.501,148.439
C00513=1234.380,110.872,-48.162,-178.261,5.502,148.438
C00514=1234.376,111.122,-48.181,-178.258,5.503,148.438
C00515=1234.371,111.371,-48.202,-178.255,5.504,148.437
C00516=1234.367,111.619,-48.221,-178.253,5.505,148.437
C00517=1234.362,111.869,-48.240,-178.251,5.506,148.436
C00518=1234.357,112.119,-48.260,-178.248,5.506,148.435
C00519=1234.352,112.367,-48.279,-178.245,5.507,148.435
C00520=1234.347,112.617,-48.299,-178.243,5.509,148.434
C00521=1234.342,112.866,-48.317,-178.240,5.509,148.434
C00522=1234.338,113.115,-48.337,-178.237,5.510,148.433
C00523=1234.333,113.365,-48.357,-178.235,5.511,148.433
C00524=1234.328,113.614,-48.376,-178.233,5.512,148.432
C00525=1234.323,113.863,-48.396,-178.229,5.513,148.431
C00526=1234.319,114.112,-48.415,-178.227,5.514,148.431
C00527=1234.313,114.361,-48.434,-178.225,5.515,148.430
C00528=1234.309,114.610,-48.454,-178.222,5.515,148.430
C00529=1234.304,114.860,-48.474,-178.220,5.516,148.429
C00530=1234.299,115.109,-48.493,-178.217,5.518,148.429
C00531=1234.294,115.358,-48.513,-178.214,5.518,148.428
C00532=1234.290,115.607,-48.532,-178.212,5.519,148.428
C00533=1234.285,115.856,-48.551,-178.210,5.520,148.427
C00534=1234.280,116.105,-48.572,-178.207,5.521,148.426
C00535=1234.276,116.355,-48.591,-178.204,5.522,148.426
C00536=1234.270,116.604,-48.611,-178.202,5.523,148.425
C00537=1234.266,116.853,-48.630,-178.199,5.524,148.425
C00538=1234.261,117.103,-48.650,-178.197,5.525,148.424
C00539=1234.256,117.351,-48.670,-178.194,5.525,148.424
C00540=1234.251,117.601,-48.690,-178.192,5.527,148.423
C00541=1234.247,117.850,-48.709,-178.189,5.528,148.423
C00542=1234.242,118.099,-48.728,-178.186,5.528,148.422
C00543=1234.237,118.348,-48.748,-178.184,5.529,148.422
C00544=1234.233,118.597,-48.768,-178.182,5.530,148.421
C00545=1234.228,118.847,-48.788,-178.179,5.532,148.421
C00546=1234.223,119.095,-48.808,-178.176,5.532,148.420
C00547=1234.218,119.345,-48.827,-178.174,5.533,148.419
C00548=1234.213,119.594,-48.847,-178.172,5.534,148.419
C00549=1234.209,119.844,-48.867,-178.168,5.535,148.418
C00550=1234.203,120.092,-48.887,-178.166,5.536,148.418
C00551=1234.199,120.342,-48.906,-178.164,5.537,148.417
C00552=1234.194,120.591,-48.927,-178.161,5.538,148.417
C00553=1234.190,120.840,-48.946,-178.159,5.539,148.416
C00554=1234.184,121.089,-48.966,-178.156,5.540,148.416
C00555=1234.180,121.338,-48.986,-178.153,5.541,148.415
C00556=1234.175,121.588,-49.006,-178.151,5.542,148.414
C00557=1234.170,121.837,-49.025,-178.149,5.542,148.414
C00558=1234.165,122.085,-49.045,-178.146,5.544,148.413
C00559=1234.161,122.335,-49.065,-178.143,5.545,148.413
C00560=1234.156,122.584,-49.085,-178.141,5.545,148.412
C00561=1234.151,122.833,-49.105,-178.139,5.546,148.412
C00562=1234.146,123.082,-49.125,-178.135,5.548,148.411
C00563=1234.142,123.331,-49.145,-178.133,5.549,148.411
C00564=1234.137,123.581,-49.164,-178.131,5.549,148.410
C00565=1234.132,123.830,-49.185,-178.128,5.550,148.409
C00566=1234.128,124.079,-49.204,-178.126,5.551,148.409
C00567=1234.123,124.328,-49.225,-178.123,5.553,148.408
C00568=1234.118,124.577,-49.244,-178.121,5.554,148.408
C00569=1234.113,124.826,-49.265,-178.118,5.554,148.407
C00570=1234.108,125.076,-49.285,-178.115,5.555,148.407
C00571=1234.103,125.325,-49.305,-178.113,5.557,148.406
C00572=1234.099,125.574,-49.325,-178.110,5.557,148.406
C00573=1234.094,125.823,-49.345,-178.108,5.558,148.405
C00574=1234.089,126.072,-49.365,-178.105,5.559,148.405
C00575=1234.085,126.321,-49.385,-178.102,5.560,148.404
C00576=1234.080,126.570,-49.405,-178.100,5.561,148.404
C00577=1234.075,126.820,-49.425,-178.098,5.562,148.403
C00578=1234.070,127.069,-49.446,-178.095,5.564,148.403
C00579=1234.066,127.318,-49.466,-178.092,5.564,148.402
C00580=1234.060,127.567,-49.485,-178.090,5.565,148.401
C00581=1234.056,127.816,-49.506,-178.088,5.566,148.401
C00582=1234.051,128.065,-49.525,-178.084,5.568,148.400
C00583=1234.047,128.314,-49.546,-178.082,5.569,148.400
C00584=1234.042,128.564,-49.567,-178.080,5.569,148.399
C00585=1234.037,128.813,-49.586,-178.078,5.570,148.399
C00586=1234.032,129.062,-49.607,-178.074,5.572,148.398
C00587=1234.028,129.311,-49.627,-178.072,5.572,148.398
C00588=1234.023,129.560,-49.646,-178.070,5.573,148.397
C00589=1234.017,129.809,-49.667,-178.067,5.574,148.397
C00590=1234.013,130.058,-49.688,-178.064,5.576,148.396
C00591=1234.008,130.308,-49.707,-178.062,5.576,148.396
C00592=1234.004,130.557,-49.728,-178.060,5.577,148.395
C00593=1233.999,130.806,-49.749,-178.056,5.579,148.395
C00594=1233.994,131.055,-49.769,-178.054,5.579,148.394
C00595=1233.989,131.304,-49.789,-178.052,5.580,148.394
C00596=1233.985,131.553,-49.809,-178.049,5.581,148.393
C00597=1233.980,131.803,-49.830,-178.047,5.583,148.393
C00598=1233.975,132.052,-49.851,-178.044,5.584,148.392
C00599=1233.971,132.301,-49.870,-178.042,5.585,148.391
C00600=1233.966,132.550,-49.891,-178.039,5.586,148.391
C00601=1233.960,132.799,-49.911,-178.037,5.587,148.390
C00602=1233.956,133.048,-49.932,-178.034,5.588,148.390
C00603=1233.952,133.297,-49.952,-178.031,5.589,148.389
C00604=1233.947,133.566,-49.974,-178.029,5.590,148.389
C00605=1233.941,133.835,-49.996,-178.026,5.591,148.388
C00606=1233.936,134.104,-50.018,-178.023,5.592,148.388
C00607=1233.931,134.372,-50.040,-178.021,5.593,148.387
C00608=1233.926,134.621,-50.061,-178.018,5.595,148.387
C00609=1233.921,134.870,-50.081,-178.015,5.595,148.386
C00610=1233.917,135.119,-50.102,-178.013,5.596,148.386
C00611=1233.912,135.368,-50.123,-178.010,5.598,148.385
C00612=1233.907,135.617,-50.143,-178.008,5.599,148.385
C00613=1233.903,135.866,-50.163,-178.005,5.599,148.384
C00614=1233.897,136.116,-50.184,-178.002,5.601,148.384
C00615=1233.893,136.365,-50.204,-178.000,5.602,148.383
C00616=1233.888,136.614,-50.225,-177.998,5.603,148.382
C00617=1233.883,136.863,-50.245,-177.994,5.604,148.382
C00618=1233.879,137.112,-50.266,-177.992,5.605,148.381
C00619=1233.874,137.361,-50.287,-177.990,5.606,148.381
C00620=1233.869,137.610,-50.307,-177.988,5.607,148.380
C00621=1233.864,137.859,-50.328,-177.985,5.608,148.380
C00622=1233.860,138.108,-50.348,-177.982,5.609,148.379
C00623=1233.855,138.357,-50.369,-177.980,5.610,148.379
C00624=1233.851,138.607,-50.390,-177.977,5.612,148.378
C00625=1233.846,138.856,-50.410,-177.975,5.613,148.378
C00626=1233.841,139.105,-50.431,-177.972,5.613,148.377
C00627=1233.837,139.354,-50.452,-177.969,5.615,148.377
C00628=1233.831,139.604,-50.473,-177.967,5.616,148.376
C00629=1233.827,139.853,-50.493,-177.965,5.617,148.376
C00630=1233.822,140.101,-50.515,-177.961,5.618,148.375
C00631=1233.818,140.350,-50.535,-177.959,5.619,148.375
C00632=1233.813,140.599,-50.556,-177.957,5.620,148.374
C00633=1233.808,140.848,-50.576,-177.954,5.622,148.374
C00634=1233.803,141.098,-50.597,-177.951,5.622,148.373
C00635=1233.798,141.347,-50.618,-177.949,5.623,148.373
C00636=1233.793,141.596,-50.639,-177.946,5.625,148.372
C00637=1233.789,141.845,-50.659,-177.944,5.626,148.372
C00638=1233.784,142.095,-50.680,-177.941,5.627,148.371
C00639=1233.780,142.343,-50.702,-177.939,5.628,148.371
C00640=1233.775,142.592,-50.723,-177.936,5.629,148.370
C00641=1233.771,142.841,-50.743,-177.934,5.631,148.370
C00642=1233.765,143.090,-50.764,-177.931,5.631,148.369
C00643=1233.761,143.339,-50.784,-177.929,5.632,148.369
C00644=1233.756,143.588,-50.806,-177.926,5.634,148.368
C00645=1233.751,143.837,-50.827,-177.924,5.635,148.368
C00646=1233.746,144.086,-50.847,-177.921,5.635,148.367
C00647=1233.742,144.336,-50.869,-177.918,5.637,148.367
C00648=1233.738,144.585,-50.890,-177.916,5.638,148.366
C00649=1233.733,144.834,-50.911,-177.914,5.639,148.366
C00650=1233.728,145.083,-50.931,-177.910,5.640,148.365
C00651=1233.723,145.332,-50.952,-177.908,5.641,148.365
C00652=1233.718,145.581,-50.974,-177.905,5.643,148.364
C00653=1233.714,145.830,-50.994,-177.903,5.644,148.364
C00654=1233.709,146.080,-51.015,-177.901,5.645,148.363
C00655=1233.704,146.328,-51.037,-177.898,5.646,148.363
C00656=1233.700,146.577,-51.057,-177.896,5.647,148.362
C00657=1233.695,146.826,-51.078,-177.893,5.648,148.362
C00658=1233.690,147.075,-51.100,-177.890,5.650,148.361
C00659=1233.686,147.325,-51.121,-177.888,5.650,148.361
C00660=1233.681,147.574,-51.142,-177.885,5.652,148.360
C00661=1233.676,147.823,-51.163,-177.883,5.653,148.360
C00662=1233.671,148.072,-51.184,-177.880,5.654,148.359
C00663=1233.666,148.321,-51.205,-177.877,5.655,148.359
C00664=1233.661,148.569,-51.226,-177.875,5.656,148.358
C00665=1233.658,148.819,-51.247,-177.873,5.657,148.358
C00666=1233.653,149.068,-51.269,-177.870,5.659,148.357
C00667=1233.647,149.317,-51.290,-177.867,5.660,148.357
C00668=1233.643,149.566,-51.310,-177.865,5.661,148.356
C00669=1233.639,149.815,-51.332,-177.863,5.662,148.356
C00670=1233.634,150.065,-51.353,-177.860,5.663,148.355
C00671=1233.629,150.313,-51.375,-177.857,5.665,148.355
C00672=1233.624,150.562,-51.395,-177.855,5.666,148.354
C00673=1233.619,150.811,-51.417,-177.852,5.667,148.354
C00674=1233.615,151.061,-51.438,-177.850,5.668,148.353
C00675=1233.610,151.309,-51.460,-177.847,5.669,148.353
C00676=1233.606,151.558,-51.480,-177.844,5.670,148.352
C00677=1233.601,151.807,-51.502,-177.842,5.671,148.352
C00678=1233.596,152.057,-51.523,-177.839,5.673,148.351
C00679=1233.591,152.306,-51.545,-177.837,5.674,148.351
C00680=1233.586,152.555,-51.566,-177.835,5.675,148.350
C00681=1233.583,152.804,-51.587,-177.832,5.676,148.350
C00682=1233.578,153.053,-51.609,-177.830,5.677,148.349
C00683=1233.572,153.302,-51.630,-177.826,5.679,148.349
C00684=1233.568,153.550,-51.652,-177.824,5.680,148.348
C00685=1233.563,153.800,-51.673,-177.821,5.681,148.348
C00686=1233.558,154.049,-51.695,-177.819,5.682,148.347
C00687=1233.554,154.297,-51.716,-177.817,5.683,148.347
C00688=1233.549,154.547,-51.737,-177.814,5.685,148.346
C00689=1233.545,154.796,-51.759,-177.812,5.686,148.346
C00690=1233.539,155.045,-51.780,-177.809,5.687,148.345
C00691=1233.535,155.294,-51.802,-177.806,5.688,148.345
C00692=1233.530,155.543,-51.824,-177.804,5.689,148.344
C00693=1233.525,155.792,-51.845,-177.801,5.691,148.344
C00694=1233.520,156.041,-51.866,-177.799,5.692,148.344
C00695=1233.516,156.290,-51.888,-177.796,5.693,148.343
C00696=1233.512,156.539,-51.909,-177.794,5.694,148.343
C00697=1233.507,156.788,-51.930,-177.791,5.696,148.342
C00698=1233.502,157.037,-51.952,-177.789,5.697,148.342
C00699=1233.498,157.286,-51.974,-177.785,5.698,148.341
C00700=1233.492,157.535,-51.995,-177.783,5.699,148.341
C00701=1233.488,157.785,-52.017,-177.781,5.700,148.340
C00702=1233.483,158.033,-52.039,-177.778,5.702,148.340
C00703=1233.479,158.283,-52.061,-177.776,5.703,148.339
C00704=1233.474,158.531,-52.083,-177.773,5.704,148.339
C00705=1233.469,158.781,-52.104,-177.771,5.705,148.338
C00706=1233.465,159.030,-52.126,-177.768,5.707,148.338
C00707=1233.460,159.278,-52.147,-177.765,5.708,148.337
C00708=1233.455,159.548,-52.170,-177.763,5.710,148.337
C00709=1233.450,159.816,-52.194,-177.760,5.710,148.336
C00710=1233.444,160.086,-52.217,-177.757,5.712,148.336
C00711=1233.440,160.355,-52.240,-177.754,5.714,148.335
C00712=1233.435,160.604,-52.262,-177.752,5.714,148.335
C00713=1233.430,160.853,-52.284,-177.749,5.716,148.334
C00714=1233.426,161.102,-52.306,-177.747,5.717,148.334
C00715=1233.421,161.351,-52.328,-177.744,5.719,148.333
C00716=1233.416,161.600,-52.350,-177.742,5.720,148.333
C00717=1233.411,161.849,-52.372,-177.739,5.720,148.332
C00718=1233.407,162.098,-52.394,-177.737,5.722,148.332
C00719=1233.402,162.347,-52.416,-177.735,5.723,148.332
C00720=1233.397,162.596,-52.437,-177.731,5.725,148.331
C00721=1233.393,162.845,-52.459,-177.729,5.726,148.331
C00722=1233.388,163.094,-52.480,-177.727,5.728,148.330
C00723=1233.383,163.343,-52.502,-177.724,5.728,148.330
C00724=1233.379,163.592,-52.524,-177.721,5.730,148.329
C00725=1233.374,163.841,-52.546,-177.719,5.731,148.329
C00726=1233.370,164.090,-52.568,-177.716,5.733,148.328
C00727=1233.365,164.339,-52.590,-177.714,5.734,148.328
C00728=1233.360,164.588,-52.612,-177.711,5.735,148.327
C00729=1233.355,164.837,-52.634,-177.709,5.736,148.327
C00730=1233.351,165.086,-52.657,-177.706,5.738,148.327
C00731=1233.346,165.334,-52.678,-177.704,5.739,148.326
C00732=1233.342,165.584,-52.700,-177.701,5.740,148.326
C00733=1233.337,165.832,-52.722,-177.698,5.741,148.325
C00734=1233.333,166.082,-52.744,-177.696,5.743,148.325
C00735=1233.328,166.330,-52.766,-177.694,5.744,148.324
C00736=1233.323,166.580,-52.788,-177.690,5.745,148.324
C00737=1233.318,166.829,-52.810,-177.688,5.746,148.323
C00738=1233.314,167.078,-52.832,-177.686,5.748,148.323
C00739=1233.309,167.327,-52.854,-177.683,5.749,148.322
C00740=1233.305,167.576,-52.876,-177.680,5.751,148.322
C00741=1233.299,167.824,-52.899,-177.678,5.752,148.322
C00742=1233.295,168.074,-52.921,-177.675,5.753,148.321
C00743=1233.290,168.322,-52.943,-177.673,5.754,148.321
C00744=1233.286,168.572,-52.965,-177.670,5.756,148.320
C00745=1233.281,168.820,-52.986,-177.668,5.757,148.320
C00746=1233.276,169.070,-53.009,-177.665,5.759,148.319
C00747=1233.271,169.318,-53.031,-177.663,5.760,148.319
C00748=1233.267,169.567,-53.053,-177.660,5.761,148.318
C00749=1233.263,169.817,-53.075,-177.658,5.762,148.318
C00750=1233.257,170.066,-53.098,-177.655,5.764,148.317
C00751=1233.253,170.314,-53.121,-177.653,5.765,148.317
C00752=1233.248,170.563,-53.142,-177.650,5.767,148.317
C00753=1233.243,170.813,-53.165,-177.647,5.767,148.316
C00754=1233.239,171.061,-53.187,-177.645,5.769,148.316
C00755=1233.235,171.310,-53.209,-177.643,5.770,148.315
C00756=1233.230,171.559,-53.231,-177.640,5.772,148.315
C00757=1233.225,171.808,-53.254,-177.637,5.773,148.314
C00758=1233.221,172.057,-53.276,-177.635,5.774,148.314
C00759=1233.216,172.306,-53.298,-177.632,5.775,148.313
C00760=1233.211,172.555,-53.321,-177.630,5.777,148.313
C00761=1233.206,172.803,-53.343,-177.627,5.778,148.313
C00762=1233.202,173.053,-53.365,-177.625,5.780,148.312
C00763=1233.197,173.302,-53.388,-177.622,5.781,148.312
C00764=1233.193,173.550,-53.410,-177.620,5.782,148.311
C00765=1233.188,173.800,-53.433,-177.617,5.784,148.311
C00766=1233.183,174.049,-53.455,-177.614,5.785,148.310
C00767=1233.179,174.297,-53.477,-177.612,5.787,148.310
C00768=1233.174,174.547,-53.500,-177.610,5.788,148.309
C00769=1233.169,174.795,-53.522,-177.606,5.789,148.309
C00770=1233.165,175.044,-53.544,-177.604,5.790,148.309
C00771=1233.160,175.294,-53.567,-177.602,5.792,148.308
C00772=1233.155,175.542,-53.589,-177.599,5.793,148.308
C00773=1233.150,175.792,-53.612,-177.596,5.795,148.307
C00774=1233.146,176.040,-53.635,-177.594,5.796,148.307
C00775=1233.141,176.289,-53.657,-177.591,5.797,148.306
C00776=1233.137,176.538,-53.680,-177.589,5.799,148.306
C00777=1233.132,176.787,-53.702,-177.587,5.800,148.306
C00778=1233.127,177.036,-53.725,-177.584,5.802,148.305
C00779=1233.123,177.285,-53.747,-177.581,5.802,148.305
C00780=1233.118,177.534,-53.770,-177.579,5.804,148.304
C00781=1233.113,177.783,-53.792,-177.577,5.805,148.304
C00782=1233.109,178.032,-53.815,-177.573,5.807,148.303
C00783=1233.105,178.280,-53.838,-177.571,5.809,148.303
C00784=1233.100,178.530,-53.861,-177.569,5.810,148.302
C00785=1233.095,178.778,-53.883,-177.566,5.812,148.302
C00786=1233.090,179.028,-53.906,-177.563,5.812,148.302
C00787=1233.086,179.277,-53.929,-177.561,5.814,148.301
C00788=1233.081,179.525,-53.952,-177.559,5.815,148.301
C00789=1233.077,179.774,-53.974,-177.556,5.817,148.300
C00790=1233.072,180.023,-53.997,-177.553,5.818,148.300
C00791=1233.068,180.273,-54.019,-177.551,5.819,148.299
C00792=1233.062,180.521,-54.042,-177.548,5.821,148.299
C00793=1233.058,180.770,-54.065,-177.546,5.822,148.298
C00794=1233.053,181.019,-54.087,-177.543,5.824,148.298
C00795=1233.049,181.268,-54.111,-177.540,5.826,148.298
C00796=1233.044,181.516,-54.133,-177.538,5.826,148.297
C00797=1233.039,181.766,-54.156,-177.535,5.828,148.297
C00798=1233.035,182.015,-54.179,-177.533,5.829,148.296
C00799=1233.030,182.264,-54.202,-177.530,5.831,148.296
C00800=1233.026,182.512,-54.224,-177.527,5.833,148.296
C00801=1233.021,182.761,-54.247,-177.525,5.834,148.295
C00802=1233.016,183.010,-54.270,-177.522,5.835,148.295
C00803=1233.012,183.259,-54.293,-177.520,5.836,148.294
C00804=1233.007,183.508,-54.316,-177.517,5.838,148.294
C00805=1233.002,183.757,-54.339,-177.515,5.840,148.293
C00806=1232.998,184.006,-54.362,-177.513,5.841,148.293
C00807=1232.993,184.255,-54.385,-177.510,5.843,148.293
C00808=1232.989,184.504,-54.408,-177.507,5.843,148.292
C00809=1232.984,184.752,-54.431,-177.505,5.845,148.292
C00810=1232.979,185.001,-54.454,-177.502,5.847,148.291
C00811=1232.974,185.251,-54.477,-177.500,5.848,148.291
C00812=1232.970,185.520,-54.501,-177.497,5.850,148.290
C00813=1232.965,185.789,-54.527,-177.494,5.851,148.290
C00814=1232.959,186.059,-54.552,-177.491,5.853,148.290
C00815=1232.955,186.328,-54.576,-177.488,5.855,148.289
C00816=1232.950,186.578,-54.600,-177.486,5.856,148.289
C00817=1232.945,186.827,-54.623,-177.483,5.857,148.288
C00818=1232.941,187.076,-54.645,-177.481,5.858,148.288
C00819=1232.936,187.325,-54.668,-177.478,5.860,148.288
C00820=1232.932,187.574,-54.692,-177.476,5.862,148.287
C00821=1232.926,187.822,-54.715,-177.473,5.863,148.287
C00822=1232.922,188.071,-54.738,-177.471,5.865,148.286
C00823=1232.918,188.320,-54.761,-177.468,5.866,148.286
C00824=1232.913,188.569,-54.784,-177.466,5.867,148.286
C00825=1232.908,188.818,-54.808,-177.463,5.869,148.285
C00826=1232.904,189.067,-54.830,-177.461,5.870,148.285
C00827=1232.900,189.316,-54.854,-177.458,5.872,148.284
C00828=1232.895,189.565,-54.877,-177.455,5.874,148.284
C00829=1232.890,189.813,-54.900,-177.453,5.875,148.283
C00830=1232.885,190.062,-54.923,-177.450,5.876,148.283
C00831=1232.881,190.311,-54.946,-177.448,5.878,148.283
C00832=1232.876,190.560,-54.970,-177.445,5.879,148.282
C00833=1232.872,190.809,-54.993,-177.443,5.881,148.282
C00834=1232.867,191.058,-55.016,-177.440,5.882,148.281
C00835=1232.863,191.306,-55.040,-177.438,5.883,148.281
C00836=1232.858,191.556,-55.064,-177.435,5.885,148.281
C00837=1232.854,191.804,-55.086,-177.432,5.887,148.280
C00838=1232.849,192.053,-55.110,-177.430,5.888,148.280
C00839=1232.844,192.302,-55.133,-177.427,5.890,148.279
C00840=1232.840,192.551,-55.157,-177.424,5.892,148.279
C00841=1232.834,192.800,-55.180,-177.422,5.893,148.279
C00842=1232.830,193.049,-55.203,-177.420,5.894,148.278
C00843=1232.825,193.297,-55.227,-177.417,5.896,148.278
C00844=1232.821,193.546,-55.250,-177.415,5.897,148.277
C00845=1232.816,193.795,-55.274,-177.412,5.899,148.277
C00846=1232.812,194.044,-55.296,-177.409,5.901,148.277
C00847=1232.807,194.293,-55.320,-177.407,5.902,148.276
C00848=1232.803,194.541,-55.344,-177.405,5.904,148.276
C00849=1232.798,194.790,-55.367,-177.401,5.905,148.275
C00850=1232.794,195.039,-55.391,-177.399,5.906,148.275
C00851=1232.789,195.288,-55.414,-177.397,5.908,148.275
C00852=1232.784,195.537,-55.438,-177.394,5.910,148.274
C00853=1232.780,195.786,-55.461,-177.392,5.911,148.274
C00854=1232.775,196.035,-55.485,-177.389,5.913,148.273
C00855=1232.770,196.284,-55.508,-177.386,5.914,148.273
C00856=1232.766,196.532,-55.532,-177.384,5.915,148.273
C00857=1232.761,196.781,-55.556,-177.381,5.917,148.272
C00858=1232.757,197.030,-55.579,-177.379,5.919,148.272
C00859=1232.752,197.279,-55.603,-177.377,5.920,148.271
C00860=1232.747,197.528,-55.626,-177.374,5.922,148.271
C00861=1232.743,197.777,-55.650,-177.371,5.923,148.271
C00862=1232.738,198.025,-55.674,-177.369,5.924,148.270
C00863=1232.734,198.274,-55.697,-177.366,5.926,148.270
C00864=1232.729,198.523,-55.721,-177.364,5.928,148.270
C00865=1232.725,198.772,-55.745,-177.361,5.930,148.269
C00866=1232.720,199.021,-55.768,-177.358,5.931,148.269
C00867=1232.715,199.269,-55.792,-177.356,5.933,148.268
C00868=1232.711,199.519,-55.816,-177.353,5.934,148.268
C00869=1232.707,199.767,-55.840,-177.351,5.935,148.268
C00870=1232.702,200.017,-55.864,-177.348,5.937,148.267
C00871=1232.697,200.265,-55.888,-177.346,5.939,148.267
C00872=1232.692,200.514,-55.911,-177.343,5.940,148.266
C00873=1232.688,200.763,-55.935,-177.341,5.942,148.266
C00874=1232.683,201.012,-55.959,-177.338,5.944,148.266
C00875=1232.679,201.261,-55.982,-177.335,5.945,148.265
C00876=1232.674,201.509,-56.006,-177.333,5.946,148.265
C00877=1232.670,201.758,-56.029,-177.331,5.948,148.265
C00878=1232.665,202.006,-56.053,-177.328,5.950,148.264
C00879=1232.660,202.255,-56.078,-177.325,5.952,148.264
C00880=1232.656,202.505,-56.102,-177.323,5.953,148.263
C00881=1232.652,202.753,-56.126,-177.320,5.955,148.263
C00882=1232.647,203.002,-56.149,-177.318,5.956,148.263
C00883=1232.642,203.251,-56.173,-177.315,5.957,148.262
C00884=1232.638,203.500,-56.197,-177.313,5.959,148.262
C00885=1232.633,203.749,-56.221,-177.310,5.961,148.262
C00886=1232.628,203.997,-56.245,-177.307,5.963,148.261
C00887=1232.623,204.246,-56.269,-177.305,5.964,148.261
C00888=1232.620,204.495,-56.293,-177.302,5.966,148.260
C00889=1232.615,204.744,-56.317,-177.300,5.967,148.260
C00890=1232.610,204.993,-56.341,-177.297,5.969,148.260
C00891=1232.605,205.241,-56.365,-177.295,5.970,148.259
C00892=1232.601,205.490,-56.389,-177.292,5.972,148.259
C00893=1232.596,205.739,-56.413,-177.289,5.974,148.258
C00894=1232.593,205.988,-56.437,-177.287,5.976,148.258
C00895=1232.587,206.237,-56.462,-177.285,5.977,148.258
C00896=1232.583,206.486,-56.485,-177.282,5.979,148.257
C00897=1232.578,206.734,-56.509,-177.279,5.980,148.257
C00898=1232.573,206.983,-56.534,-177.277,5.982,148.257
C00899=1232.569,207.232,-56.558,-177.275,5.983,148.256
C00900=1232.565,207.481,-56.582,-177.272,5.985,148.256
C00901=1232.560,207.729,-56.606,-177.269,5.987,148.256
C00902=1232.555,207.978,-56.631,-177.266,5.989,148.255
C00903=1232.551,208.226,-56.655,-177.264,5.990,148.255
C00904=1232.547,208.476,-56.678,-177.261,5.991,148.254
C00905=1232.542,208.725,-56.703,-177.259,5.993,148.254
C00906=1232.537,208.973,-56.727,-177.256,5.995,148.254
C00907=1232.533,209.222,-56.751,-177.254,5.996,148.253
C00908=1232.528,209.470,-56.776,-177.252,5.998,148.253
C00909=1232.524,209.720,-56.800,-177.249,6.000,148.253
C00910=1232.519,209.969,-56.824,-177.246,6.002,148.252
C00911=1232.514,210.217,-56.848,-177.243,6.003,148.252
C00912=1232.510,210.466,-56.872,-177.241,6.004,148.251
C00913=1232.505,210.715,-56.897,-177.238,6.006,148.251
C00914=1232.501,210.964,-56.922,-177.236,6.008,148.251
C00915=1232.496,211.212,-56.946,-177.233,6.010,148.250
C00916=1232.491,211.482,-56.972,-177.231,6.012,148.250
C00917=1232.486,211.754,-56.999,-177.228,6.014,148.250
C00918=1232.481,212.024,-57.025,-177.225,6.015,148.249
C00919=1232.476,212.294,-57.052,-177.222,6.017,148.249
C00920=1232.472,212.542,-57.076,-177.220,6.019,148.248
C00921=1232.468,212.792,-57.101,-177.217,6.020,148.248
C00922=1232.463,213.040,-57.125,-177.215,6.022,148.248
C00923=1232.458,213.289,-57.149,-177.212,6.024,148.247
C00924=1232.454,213.538,-57.174,-177.210,6.026,148.247
C00925=1232.449,213.786,-57.198,-177.207,6.027,148.247
C00926=1232.444,214.035,-57.223,-177.204,6.028,148.246
C00927=1232.440,214.284,-57.247,-177.202,6.030,148.246
C00928=1232.435,214.533,-57.272,-177.199,6.032,148.245
C00929=1232.431,214.781,-57.296,-177.197,6.034,148.245
C00930=1232.426,215.030,-57.321,-177.194,6.036,148.245
C00931=1232.422,215.279,-57.345,-177.192,6.037,148.244
C00932=1232.417,215.528,-57.370,-177.189,6.039,148.244
C00933=1232.412,215.776,-57.394,-177.187,6.040,148.244
C00934=1232.408,216.025,-57.420,-177.184,6.042,148.243
C00935=1232.404,216.274,-57.444,-177.181,6.044,148.243
C00936=1232.399,216.522,-57.469,-177.179,6.045,148.243
C00937=1232.395,216.771,-57.493,-177.177,6.047,148.242
C00938=1232.390,217.020,-57.518,-177.174,6.049,148.242
C00939=1232.385,217.270,-57.543,-177.171,6.051,148.242
C00940=1232.381,217.517,-57.568,-177.169,6.053,148.241
C00941=1232.376,217.766,-57.592,-177.166,6.054,148.241
C00942=1232.372,218.015,-57.617,-177.164,6.055,148.241
C00943=1232.367,218.264,-57.641,-177.161,6.057,148.240
C00944=1232.362,218.513,-57.666,-177.158,6.059,148.240
C00945=1232.359,218.761,-57.691,-177.156,6.061,148.240
C00946=1232.353,219.010,-57.716,-177.153,6.063,148.239
C00947=1232.350,219.259,-57.740,-177.151,6.064,148.239
C00948=1232.344,219.508,-57.765,-177.148,6.066,148.239
C00949=1232.340,219.756,-57.790,-177.146,6.067,148.238
C00950=1232.336,220.005,-57.815,-177.143,6.069,148.238
C00951=1232.331,220.254,-57.839,-177.140,6.071,148.238
C00952=1232.326,220.503,-57.865,-177.138,6.073,148.237
C00953=1232.322,220.751,-57.889,-177.136,6.074,148.237
C00954=1232.318,221.000,-57.914,-177.133,6.076,148.237
C00955=1232.313,221.248,-57.940,-177.131,6.078,148.236
C00956=1232.308,221.497,-57.964,-177.128,6.080,148.236
C00957=1232.304,221.746,-57.989,-177.125,6.082,148.236
C00958=1232.299,221.994,-58.014,-177.123,6.083,148.235
C00959=1232.295,222.243,-58.039,-177.121,6.084,148.235
C00960=1232.290,222.492,-58.063,-177.118,6.086,148.235
C00961=1232.286,222.741,-58.089,-177.115,6.088,148.234
C00962=1232.281,222.990,-58.114,-177.113,6.090,148.234
C00963=1232.277,223.238,-58.139,-177.110,6.092,148.234
C00964=1232.272,223.487,-58.164,-177.107,6.094,148.233
C00965=1232.268,223.736,-58.189,-177.105,6.096,148.233
C00966=1232.263,223.984,-58.214,-177.103,6.097,148.233
C00967=1232.259,224.233,-58.239,-177.100,6.099,148.232
C00968=1232.254,224.482,-58.264,-177.098,6.100,148.232
C00969=1232.250,224.731,-58.289,-177.095,6.102,148.232
C00970=1232.245,224.979,-58.314,-177.092,6.104,148.231
C00971=1232.241,225.228,-58.339,-177.090,6.106,148.231
C00972=1232.236,225.476,-58.364,-177.088,6.107,148.231
C00973=1232.232,225.725,-58.390,-177.085,6.109,148.230
C00974=1232.227,225.974,-58.414,-177.082,6.111,148.230
C00975=1232.223,226.223,-58.440,-177.080,6.113,148.230
C00976=1232.217,226.472,-58.465,-177.077,6.115,148.229
C00977=1232.214,226.720,-58.490,-177.075,6.117,148.229
C00978=1232.209,226.969,-58.515,-177.072,6.118,148.229
C00979=1232.205,227.218,-58.540,-177.070,6.119,148.228
C00980=1232.200,227.466,-58.566,-177.067,6.121,148.228
C00981=1232.195,227.715,-58.591,-177.065,6.123,148.228
C00982=1232.191,227.964,-58.617,-177.062,6.125,148.227
C00983=1232.186,228.213,-58.641,-177.059,6.127,148.227
C00984=1232.182,228.461,-58.666,-177.057,6.129,148.227
C00985=1232.178,228.709,-58.692,-177.054,6.131,148.226
C00986=1232.173,228.959,-58.717,-177.051,6.133,148.226
C00987=1232.168,229.207,-58.742,-177.049,6.134,148.226
C00988=1232.164,229.456,-58.768,-177.047,6.135,148.225
C00989=1232.160,229.704,-58.794,-177.044,6.137,148.225
C00990=1232.155,229.953,-58.818,-177.042,6.140,148.225
C00991=1232.150,230.202,-58.844,-177.039,6.141,148.225
C00992=1232.146,230.450,-58.870,-177.037,6.143,148.224
C00993=1232.141,230.699,-58.895,-177.034,6.145,148.224
C00994=1232.137,230.948,-58.920,-177.032,6.146,148.224
C00995=1232.132,231.196,-58.946,-177.029,6.148,148.223
C00996=1232.128,231.445,-58.972,-177.027,6.150,148.223
C00997=1232.123,231.693,-58.997,-177.024,6.152,148.223
C00998=1232.118,231.943,-59.022,-177.022,6.154,148.222
C00999=1232.114,232.191,-59.048,-177.019,6.156,148.222
C01000=1232.109,232.440,-59.073,-177.016,6.157,148.222
C01001=1232.105,232.688,-59.099,-177.014,6.159,148.221
C01002=1232.101,232.937,-59.125,-177.011,6.161,148.221
C01003=1232.096,233.185,-59.150,-177.009,6.162,148.221
C01004=1232.092,233.435,-59.175,-177.006,6.164,148.220
C01005=1232.087,233.683,-59.200,-177.004,6.166,148.220
C01006=1232.082,233.932,-59.226,-177.002,6.168,148.220
C01007=1232.078,234.180,-59.252,-176.999,6.170,148.220
C01008=1232.073,234.428,-59.277,-176.997,6.172,148.219
C01009=1232.069,234.677,-59.303,-176.994,6.174,148.219
C01010=1232.065,234.926,-59.329,-176.991,6.176,148.219
C01011=1232.060,235.174,-59.354,-176.989,6.178,148.218
C01012=1232.056,235.423,-59.380,-176.987,6.179,148.218
C01013=1232.052,235.672,-59.406,-176.984,6.181,148.218
C01014=1232.047,235.921,-59.431,-176.981,6.182,148.217
C01015=1232.043,236.169,-59.457,-176.979,6.184,148.217
C01016=1232.038,236.418,-59.483,-176.976,6.186,148.217
C01017=1232.033,236.667,-59.509,-176.974,6.188,148.217
C01018=1232.029,236.915,-59.534,-176.971,6.190,148.216
C01019=1232.024,237.164,-59.560,-176.969,6.192,148.216
C01020=1232.020,237.435,-59.588,-176.966,6.194,148.216
C01021=1232.014,237.707,-59.616,-176.964,6.196,148.215
C01022=1232.010,237.978,-59.644,-176.961,6.198,148.215
C01023=1232.005,238.249,-59.672,-176.958,6.200,148.215
C01024=1232.001,238.498,-59.698,-176.956,6.202,148.214
C01025=1231.996,238.747,-59.724,-176.953,6.203,148.214
C01026=1231.991,238.996,-59.750,-176.950,6.205,148.214
C01027=1231.987,239.244,-59.775,-176.948,6.207,148.213
C01028=1231.982,239.493,-59.801,-176.945,6.209,148.213
C01029=1231.978,239.741,-59.828,-176.943,6.211,148.213
C01030=1231.974,239.990,-59.853,-176.940,6.213,148.213
C01031=1231.969,240.238,-59.879,-176.938,6.215,148.212
C01032=1231.964,240.487,-59.905,-176.935,6.217,148.212
C01033=1231.960,240.736,-59.931,-176.933,6.219,148.212
C01034=1231.956,240.985,-59.957,-176.930,6.221,148.212
C01035=1231.951,241.232,-59.983,-176.927,6.223,148.211
C01036=1231.946,241.481,-60.009,-176.925,6.224,148.211
C01037=1231.942,241.730,-60.035,-176.923,6.226,148.211
C01038=1231.938,241.979,-60.061,-176.921,6.228,148.210
C01039=1231.933,242.227,-60.088,-176.918,6.230,148.210
C01040=1231.928,242.475,-60.113,-176.915,6.231,148.210
C01041=1231.924,242.724,-60.139,-176.913,6.233,148.210
C01042=1231.919,242.973,-60.165,-176.910,6.235,148.209
C01043=1231.915,243.221,-60.192,-176.908,6.237,148.209
C01044=1231.911,243.470,-60.217,-176.905,6.239,148.209
C01045=1231.906,243.719,-60.244,-176.903,6.241,148.208
C01046=1231.902,243.967,-60.270,-176.900,6.243,148.208
C01047=1231.897,244.216,-60.296,-176.898,6.245,148.208
C01048=1231.892,244.465,-60.322,-176.895,6.247,148.208
C01049=1231.889,244.713,-60.348,-176.892,6.249,148.207
C01050=1231.884,244.962,-60.374,-176.890,6.251,148.207
C01051=1231.879,245.211,-60.400,-176.888,6.253,148.207
C01052=1231.875,245.459,-60.427,-176.886,6.254,148.206
C01053=1231.871,245.707,-60.452,-176.883,6.256,148.206
C01054=1231.866,245.956,-60.479,-176.880,6.258,148.206
C01055=1231.862,246.204,-60.505,-176.878,6.260,148.206
C01056=1231.857,246.454,-60.531,-176.875,6.261,148.205
C01057=1231.853,246.702,-60.558,-176.873,6.264,148.205
C01058=1231.849,246.951,-60.584,-176.870,6.266,148.205
C01059=1231.844,247.199,-60.611,-176.868,6.267,148.205
C01060=1231.840,247.448,-60.636,-176.865,6.269,148.204
C01061=1231.835,247.696,-60.664,-176.863,6.271,148.204
C01062=1231.830,247.944,-60.689,-176.860,6.273,148.204
C01063=1231.826,248.193,-60.716,-176.858,6.275,148.204
C01064=1231.821,248.442,-60.742,-176.855,6.277,148.203
C01065=1231.817,248.690,-60.769,-176.853,6.279,148.203
C01066=1231.813,248.939,-60.795,-176.850,6.281,148.203
C01067=1231.808,249.188,-60.822,-176.848,6.283,148.203
C01068=1231.804,249.436,-60.847,-176.845,6.285,148.202
C01069=1231.799,249.685,-60.874,-176.843,6.287,148.202
C01070=1231.795,249.933,-60.901,-176.840,6.289,148.202
C01071=1231.790,250.182,-60.927,-176.837,6.291,148.201
C01072=1231.786,250.430,-60.954,-176.835,6.293,148.201
C01073=1231.781,250.680,-60.980,-176.833,6.295,148.201
C01074=1231.777,250.928,-61.006,-176.830,6.297,148.201
C01075=1231.773,251.176,-61.034,-176.828,6.299,148.200
C01076=1231.768,251.425,-61.059,-176.825,6.301,148.200
C01077=1231.764,251.673,-61.086,-176.823,6.303,148.200
C01078=1231.759,251.921,-61.112,-176.820,6.305,148.200
C01079=1231.754,252.170,-61.139,-176.818,6.306,148.199
C01080=1231.750,252.418,-61.165,-176.815,6.309,148.199
C01081=1231.746,252.667,-61.192,-176.813,6.311,148.199
C01082=1231.741,252.916,-61.219,-176.810,6.312,148.199
C01083=1231.737,253.164,-61.245,-176.808,6.314,148.198
C01084=1231.732,253.413,-61.272,-176.805,6.316,148.198
C01085=1231.728,253.661,-61.299,-176.803,6.318,148.198
C01086=1231.723,253.910,-61.325,-176.800,6.320,148.198
C01087=1231.719,254.158,-61.352,-176.798,6.322,148.197
C01088=1231.715,254.407,-61.379,-176.795,6.324,148.197
C01089=1231.711,254.656,-61.406,-176.793,6.326,148.197
C01090=1231.706,254.904,-61.433,-176.790,6.328,148.197
C01091=1231.702,255.153,-61.459,-176.788,6.330,148.196
C01092=1231.697,255.402,-61.486,-176.786,6.332,148.196
C01093=1231.692,255.650,-61.513,-176.783,6.334,148.196
C01094=1231.689,255.898,-61.539,-176.780,6.336,148.196
C01095=1231.684,256.147,-61.566,-176.778,6.338,148.195
C01096=1231.679,256.395,-61.594,-176.776,6.340,148.195
C01097=1231.675,256.644,-61.619,-176.773,6.342,148.195
C01098=1231.670,256.893,-61.646,-176.770,6.344,148.195
C01099=1231.666,257.141,-61.673,-176.768,6.346,148.194
C01100=1231.662,257.389,-61.700,-176.766,6.348,148.194
C01101=1231.657,257.638,-61.727,-176.763,6.350,148.194
C01102=1231.652,257.886,-61.754,-176.761,6.352,148.194
C01103=1231.648,258.135,-61.781,-176.758,6.354,148.194
C01104=1231.644,258.383,-61.807,-176.756,6.356,148.193
C01105=1231.639,258.631,-61.835,-176.753,6.358,148.193
C01106=1231.635,258.881,-61.862,-176.751,6.360,148.193
C01107=1231.631,259.129,-61.889,-176.748,6.362,148.193
C01108=1231.626,259.378,-61.916,-176.746,6.364,148.192
C01109=1231.622,259.626,-61.943,-176.743,6.366,148.192
C01110=1231.617,259.874,-61.970,-176.741,6.368,148.192
C01111=1231.613,260.123,-61.997,-176.739,6.370,148.192
C01112=1231.608,260.371,-62.024,-176.736,6.372,148.191
C01113=1231.603,260.620,-62.051,-176.734,6.374,148.191
C01114=1231.600,260.869,-62.078,-176.731,6.376,148.191
C01115=1231.595,261.117,-62.105,-176.729,6.378,148.191
C01116=1231.591,261.366,-62.132,-176.727,6.380,148.190
C01117=1231.586,261.614,-62.159,-176.724,6.382,148.190
C01118=1231.581,261.863,-62.186,-176.721,6.384,148.190
C01119=1231.577,262.110,-62.214,-176.719,6.386,148.190
C01120=1231.573,262.359,-62.240,-176.717,6.388,148.190
C01121=1231.569,262.608,-62.268,-176.714,6.390,148.189
C01122=1231.564,262.856,-62.295,-176.712,6.392,148.189
C01123=1231.560,263.105,-62.322,-176.709,6.395,148.189
C01124=1231.555,263.377,-62.351,-176.706,6.396,148.189
C01125=1231.550,263.650,-62.382,-176.704,6.398,148.188
C01126=1231.545,263.922,-62.411,-176.700,6.401,148.188
C01127=1231.540,264.195,-62.441,-176.698,6.403,148.188
C01128=1231.535,264.443,-62.469,-176.696,6.405,148.188
C01129=1231.531,264.692,-62.496,-176.693,6.407,148.187
C01130=1231.527,264.941,-62.523,-176.691,6.409,148.187
C01131=1231.523,265.189,-62.550,-176.688,6.411,148.187
C01132=1231.519,265.437,-62.578,-176.686,6.413,148.187
C01133=1231.514,265.686,-62.605,-176.684,6.415,148.187
C01134=1231.510,265.935,-62.632,-176.681,6.417,148.186
C01135=1231.505,266.183,-62.659,-176.678,6.419,148.186
C01136=1231.501,266.431,-62.687,-176.676,6.422,148.186
C01137=1231.496,266.679,-62.714,-176.673,6.424,148.186
C01138=1231.492,266.929,-62.741,-176.671,6.426,148.186
C01139=1231.488,267.177,-62.769,-176.668,6.428,148.185
C01140=1231.483,267.425,-62.796,-176.666,6.430,148.185
C01141=1231.479,267.673,-62.824,-176.664,6.432,148.185
C01142=1231.475,267.922,-62.851,-176.661,6.434,148.185
C01143=1231.470,268.171,-62.878,-176.659,6.436,148.185
C01144=1231.465,268.419,-62.907,-176.656,6.438,148.184
C01145=1231.460,268.667,-62.934,-176.654,6.440,148.184
C01146=1231.457,268.916,-62.962,-176.652,6.442,148.184
C01147=1231.452,269.164,-62.989,-176.649,6.444,148.184
C01148=1231.447,269.413,-63.016,-176.646,6.447,148.184
C01149=1231.443,269.661,-63.044,-176.644,6.449,148.183
C01150=1231.439,269.910,-63.071,-176.641,6.451,148.183
C01151=1231.434,270.158,-63.099,-176.639,6.453,148.183
C01152=1231.430,270.406,-63.126,-176.637,6.455,148.183
C01153=1231.426,270.655,-63.154,-176.634,6.457,148.183
C01154=1231.421,270.903,-63.181,-176.632,6.459,148.182
C01155=1231.417,271.151,-63.209,-176.629,6.461,148.182
C01156=1231.412,271.401,-63.237,-176.627,6.463,148.182
C01157=1231.408,271.649,-63.265,-176.624,6.465,148.182
C01158=1231.403,271.897,-63.292,-176.622,6.468,148.182
C01159=1231.399,272.146,-63.320,-176.619,6.470,148.181
C01160=1231.395,272.394,-63.348,-176.617,6.473,148.181
C01161=1231.390,272.642,-63.375,-176.615,6.474,148.181
C01162=1231.386,272.891,-63.404,-176.612,6.477,148.181
C01163=1231.381,273.139,-63.431,-176.610,6.479,148.181
C01164=1231.377,273.387,-63.459,-176.607,6.480,148.180
C01165=1231.373,273.636,-63.487,-176.605,6.483,148.180
C01166=1231.369,273.884,-63.514,-176.602,6.485,148.180
C01167=1231.364,274.133,-63.543,-176.600,6.487,148.180
C01168=1231.360,274.381,-63.570,-176.597,6.490,148.180
C01169=1231.355,274.630,-63.597,-176.595,6.492,148.179
C01170=1231.351,274.878,-63.626,-176.593,6.494,148.179
C01171=1231.347,275.126,-63.653,-176.590,6.496,148.179
C01172=1231.342,275.375,-63.681,-176.588,6.498,148.179
C01173=1231.338,275.624,-63.709,-176.586,6.500,148.179
C01174=1231.333,275.871,-63.737,-176.583,6.502,148.178
C01175=1231.330,276.120,-63.765,-176.581,6.504,148.178
C01176=1231.324,276.369,-63.793,-176.578,6.507,148.178
C01177=1231.320,276.617,-63.820,-176.576,6.509,148.178
C01178=1231.316,276.865,-63.849,-176.573,6.511,148.178
C01179=1231.311,277.113,-63.877,-176.571,6.513,148.178
C01180=1231.307,277.362,-63.905,-176.568,6.515,148.177
C01181=1231.303,277.610,-63.932,-176.566,6.517,148.177
C01182=1231.298,277.859,-63.961,-176.564,6.519,148.177
C01183=1231.294,278.107,-63.989,-176.562,6.521,148.177
C01184=1231.290,278.356,-64.017,-176.558,6.524,148.177
C01185=1231.285,278.604,-64.045,-176.556,6.526,148.177
C01186=1231.281,278.852,-64.073,-176.554,6.528,148.176
C01187=1231.277,279.101,-64.100,-176.552,6.530,148.176
C01188=1231.272,279.349,-64.129,-176.549,6.532,148.176
C01189=1231.268,279.598,-64.157,-176.547,6.535,148.176
C01190=1231.263,279.846,-64.185,-176.544,6.536,148.176
C01191=1231.259,280.095,-64.213,-176.542,6.540,148.176
C01192=1231.255,280.342,-64.241,-176.539,6.541,148.175
C01193=1231.250,280.591,-64.270,-176.537,6.544,148.175
C01194=1231.246,280.839,-64.298,-176.534,6.546,148.175
C01195=1231.242,281.088,-64.326,-176.532,6.548,148.175
C01196=1231.237,281.336,-64.354,-176.530,6.550,148.175
C01197=1231.233,281.585,-64.382,-176.527,6.553,148.175
C01198=1231.228,281.833,-64.411,-176.525,6.555,148.175
C01199=1231.224,282.081,-64.439,-176.522,6.557,148.174
C01200=1231.219,282.330,-64.467,-176.520,6.559,148.174
C01201=1231.216,282.578,-64.495,-176.518,6.561,148.174
C01202=1231.211,282.826,-64.523,-176.516,6.563,148.174
C01203=1231.207,283.075,-64.552,-176.513,6.565,148.174
C01204=1231.202,283.323,-64.580,-176.510,6.568,148.174
C01205=1231.198,283.572,-64.608,-176.508,6.570,148.174
C01206=1231.194,283.820,-64.636,-176.506,6.572,148.173
C01207=1231.189,284.068,-64.665,-176.503,6.574,148.173
C01208=1231.186,284.316,-64.694,-176.501,6.576,148.173
C01209=1231.180,284.565,-64.722,-176.498,6.579,148.173
C01210=1231.176,284.813,-64.751,-176.496,6.581,148.173
C01211=1231.172,285.061,-64.779,-176.494,6.584,148.173
C01212=1231.167,285.310,-64.807,-176.491,6.586,148.172
C01213=1231.163,285.558,-64.835,-176.489,6.588,148.172
C01214=1231.159,285.806,-64.865,-176.487,6.590,148.172
C01215=1231.155,286.055,-64.893,-176.484,6.593,148.172
C01216=1231.150,286.303,-64.921,-176.481,6.595,148.172
C01217=1231.146,286.552,-64.949,-176.479,6.597,148.172
C01218=1231.141,286.800,-64.978,-176.477,6.599,148.171
C01219=1231.137,287.048,-65.007,-176.475,6.601,148.171
C01220=1231.132,287.296,-65.035,-176.473,6.603,148.171
C01221=1231.128,287.545,-65.064,-176.469,6.606,148.171
C01222=1231.124,287.793,-65.092,-176.467,6.608,148.171
C01223=1231.119,288.041,-65.121,-176.465,6.611,148.171
C01224=1231.115,288.290,-65.150,-176.463,6.613,148.171
C01225=1231.111,288.539,-65.178,-176.460,6.615,148.171
C01226=1231.106,288.786,-65.207,-176.457,6.617,148.170
C01227=1231.102,289.035,-65.236,-176.455,6.620,148.170
C01228=1231.098,289.309,-65.267,-176.453,6.622,148.170
C01229=1231.092,289.583,-65.298,-176.450,6.625,148.170
C01230=1231.088,289.857,-65.330,-176.448,6.627,148.170
C01231=1231.083,290.131,-65.362,-176.445,6.630,148.170
C01232=1231.079,290.380,-65.391,-176.443,6.632,148.170
C01233=1231.074,290.627,-65.420,-176.441,6.634,148.170
C01234=1231.070,290.876,-65.448,-176.437,6.637,148.169
C01235=1231.066,291.125,-65.477,-176.435,6.639,148.169
C01236=1231.061,291.372,-65.506,-176.433,6.641,148.169
C01237=1231.057,291.621,-65.534,-176.431,6.643,148.169
C01238=1231.053,291.869,-65.563,-176.428,6.645,148.169
C01239=1231.048,292.117,-65.592,-176.426,6.648,148.169
C01240=1231.044,292.366,-65.621,-176.423,6.650,148.169
C01241=1231.040,292.614,-65.649,-176.421,6.653,148.169
C01242=1231.035,292.862,-65.678,-176.419,6.655,148.168
C01243=1231.031,293.111,-65.707,-176.417,6.657,148.168
C01244=1231.026,293.359,-65.737,-176.414,6.660,148.168
C01245=1231.022,293.608,-65.765,-176.412,6.662,148.168
C01246=1231.018,293.855,-65.794,-176.410,6.664,148.168
C01247=1231.013,294.104,-65.823,-176.407,6.666,148.168
C01248=1231.009,294.352,-65.852,-176.405,6.668,148.168
C01249=1231.005,294.601,-65.881,-176.402,6.671,148.168
C01250=1231.000,294.849,-65.910,-176.400,6.674,148.168
C01251=1230.997,295.097,-65.939,-176.398,6.675,148.167
C01252=1230.992,295.345,-65.967,-176.395,6.678,148.167
C01253=1230.987,295.593,-65.996,-176.393,6.681,148.167
C01254=1230.983,295.841,-66.026,-176.391,6.683,148.167
C01255=1230.979,296.090,-66.055,-176.389,6.685,148.167
C01256=1230.974,296.338,-66.084,-176.386,6.687,148.167
C01257=1230.971,296.586,-66.113,-176.384,6.689,148.167
C01258=1230.966,296.835,-66.141,-176.381,6.692,148.167
C01259=1230.962,297.083,-66.171,-176.379,6.695,148.167
C01260=1230.957,297.331,-66.200,-176.377,6.697,148.167
C01261=1230.953,297.580,-66.229,-176.374,6.699,148.166
C01262=1230.948,297.828,-66.258,-176.372,6.702,148.166
C01263=1230.944,298.076,-66.288,-176.370,6.704,148.166
C01264=1230.940,298.324,-66.317,-176.368,6.706,148.166
C01265=1230.935,298.573,-66.346,-176.365,6.708,148.166
C01266=1230.931,298.821,-66.375,-176.362,6.711,148.166
C01267=1230.927,299.070,-66.405,-176.360,6.713,148.166
C01268=1230.922,299.317,-66.434,-176.358,6.716,148.166
C01269=1230.918,299.565,-66.463,-176.356,6.718,148.166
C01270=1230.914,299.814,-66.491,-176.353,6.720,148.166
C01271=1230.910,300.062,-66.521,-176.351,6.723,148.166
C01272=1230.906,300.310,-66.550,-176.349,6.725,148.166
C01273=1230.901,300.558,-66.579,-176.347,6.727,148.165
C01274=1230.897,300.806,-66.609,-176.344,6.730,148.165
C01275=1230.893,301.055,-66.638,-176.342,6.733,148.165
C01276=1230.889,301.303,-66.668,-176.340,6.735,148.165
C01277=1230.883,301.552,-66.697,-176.337,6.737,148.165
C01278=1230.879,301.800,-66.726,-176.335,6.739,148.165
C01279=1230.875,302.049,-66.756,-176.332,6.742,148.165
C01280=1230.870,302.296,-66.785,-176.330,6.744,148.165
C01281=1230.866,302.544,-66.814,-176.328,6.746,148.165
C01282=1230.862,302.793,-66.844,-176.326,6.749,148.165
C01283=1230.858,303.041,-66.873,-176.323,6.752,148.165
C01284=1230.854,303.289,-66.903,-176.321,6.754,148.165
C01285=1230.849,303.537,-66.932,-176.319,6.756,148.165
C01286=1230.845,303.786,-66.962,-176.317,6.758,148.164
C01287=1230.841,304.034,-66.991,-176.314,6.761,148.164
C01288=1230.837,304.282,-67.021,-176.312,6.763,148.164
C01289=1230.832,304.530,-67.050,-176.310,6.766,148.164
C01290=1230.828,304.778,-67.079,-176.308,6.768,148.164
C01291=1230.823,305.027,-67.109,-176.305,6.771,148.164
C01292=1230.819,305.275,-67.139,-176.303,6.773,148.164
C01293=1230.815,305.523,-67.168,-176.301,6.775,148.164
C01294=1230.810,305.771,-67.198,-176.299,6.778,148.164
C01295=1230.806,306.020,-67.227,-176.296,6.781,148.164
C01296=1230.802,306.267,-67.257,-176.293,6.783,148.164
C01297=1230.797,306.516,-67.287,-176.291,6.785,148.164
C01298=1230.793,306.764,-67.317,-176.289,6.787,148.164
C01299=1230.789,307.012,-67.346,-176.287,6.790,148.164
C01300=1230.785,307.261,-67.376,-176.284,6.792,148.164
C01301=1230.781,307.509,-67.405,-176.282,6.794,148.164
C01302=1230.776,307.758,-67.435,-176.280,6.798,148.164
C01303=1230.772,308.005,-67.465,-176.278,6.800,148.164
C01304=1230.768,308.254,-67.495,-176.276,6.802,148.164
C01305=1230.763,308.502,-67.524,-176.273,6.804,148.163
C01306=1230.759,308.750,-67.554,-176.271,6.807,148.164
C01307=1230.755,308.998,-67.584,-176.269,6.809,148.163
C01308=1230.750,309.246,-67.613,-176.267,6.812,148.163
C01309=1230.746,309.494,-67.643,-176.264,6.814,148.163
C01310=1230.742,309.742,-67.672,-176.262,6.817,148.163
C01311=1230.737,309.990,-67.703,-176.260,6.819,148.163
C01312=1230.733,310.238,-67.733,-176.258,6.821,148.163
C01313=1230.729,310.487,-67.762,-176.256,6.824,148.163
C01314=1230.725,310.735,-67.793,-176.253,6.827,148.163
C01315=1230.720,310.984,-67.823,-176.251,6.829,148.163
C01316=1230.716,311.232,-67.852,-176.249,6.831,148.163
C01317=1230.712,311.479,-67.882,-176.246,6.834,148.163
C01318=1230.707,311.728,-67.912,-176.244,6.836,148.163
C01319=1230.703,311.976,-67.942,-176.242,6.839,148.163
C01320=1230.699,312.224,-67.972,-176.240,6.841,148.163
C01321=1230.694,312.473,-68.002,-176.238,6.844,148.163
C01322=1230.690,312.721,-68.031,-176.235,6.847,148.163
C01323=1230.686,312.969,-68.062,-176.233,6.849,148.163
C01324=1230.681,313.217,-68.092,-176.231,6.851,148.163
C01325=1230.678,313.465,-68.122,-176.229,6.854,148.163
C01326=1230.673,313.713,-68.152,-176.226,6.856,148.163
C01327=1230.669,313.961,-68.182,-176.224,6.858,148.163
C01328=1230.665,314.209,-68.212,-176.222,6.862,148.163
C01329=1230.660,314.457,-68.242,-176.220,6.864,148.163
C01330=1230.656,314.705,-68.272,-176.218,6.866,148.163
C01331=1230.651,314.953,-68.302,-176.215,6.868,148.163
C01332=1230.647,315.229,-68.335,-176.213,6.871,148.163
C01333=1230.642,315.505,-68.370,-176.210,6.874,148.163
C01334=1230.637,315.781,-68.402,-176.208,6.877,148.163
C01335=1230.632,316.056,-68.437,-176.205,6.880,148.163
C01336=1230.628,316.305,-68.466,-176.204,6.882,148.163
C01337=1230.624,316.552,-68.496,-176.201,6.885,148.163
C01338=1230.620,316.802,-68.527,-176.199,6.887,148.163
C01339=1230.616,317.049,-68.557,-176.197,6.890,148.163
C01340=1230.611,317.298,-68.587,-176.195,6.892,148.163
C01341=1230.607,317.545,-68.617,-176.192,6.895,148.163
C01342=1230.603,317.793,-68.648,-176.191,6.898,148.163
C01343=1230.599,318.042,-68.677,-176.188,6.900,148.163
C01344=1230.594,318.290,-68.708,-176.186,6.903,148.163
C01345=1230.591,318.538,-68.739,-176.184,6.905,148.163
C01346=1230.586,318.787,-68.769,-176.182,6.907,148.163
C01347=1230.582,319.034,-68.799,-176.179,6.909,148.163
C01348=1230.577,319.282,-68.830,-176.177,6.913,148.163
C01349=1230.572,319.531,-68.860,-176.175,6.915,148.163
C01350=1230.568,319.778,-68.890,-176.173,6.917,148.163
C01351=1230.564,320.027,-68.921,-176.171,6.920,148.163
C01352=1230.561,320.275,-68.951,-176.169,6.923,148.163
C01353=1230.556,320.523,-68.981,-176.167,6.925,148.163
C01354=1230.552,320.771,-69.011,-176.165,6.927,148.163
C01355=1230.547,321.019,-69.042,-176.162,6.930,148.163
C01356=1230.543,321.268,-69.073,-176.160,6.933,148.163
C01357=1230.539,321.515,-69.103,-176.158,6.935,148.163
C01358=1230.534,321.764,-69.133,-176.156,6.937,148.163
C01359=1230.530,322.011,-69.164,-176.154,6.940,148.163
C01360=1230.526,322.259,-69.194,-176.152,6.943,148.163
C01361=1230.522,322.508,-69.225,-176.150,6.945,148.163
C01362=1230.518,322.756,-69.256,-176.147,6.948,148.163
C01363=1230.513,323.004,-69.286,-176.145,6.951,148.163
C01364=1230.508,323.252,-69.316,-176.143,6.953,148.163
C01365=1230.505,323.501,-69.347,-176.141,6.955,148.163
C01366=1230.501,323.749,-69.378,-176.139,6.958,148.163
C01367=1230.496,323.996,-69.408,-176.137,6.961,148.163
C01368=1230.492,324.244,-69.439,-176.135,6.963,148.163
C01369=1230.488,324.493,-69.470,-176.132,6.966,148.163
C01370=1230.483,324.741,-69.501,-176.130,6.968,148.163
C01371=1230.480,324.988,-69.531,-176.129,6.971,148.164
C01372=1230.475,325.236,-69.561,-176.127,6.973,148.164
C01373=1230.471,325.485,-69.593,-176.124,6.976,148.164
C01374=1230.467,325.733,-69.623,-176.122,6.979,148.164
C01375=1230.462,325.981,-69.654,-176.120,6.981,148.164
C01376=1230.458,326.229,-69.684,-176.118,6.984,148.164
C01377=1230.454,326.477,-69.715,-176.116,6.987,148.164
C01378=1230.450,326.725,-69.746,-176.114,6.989,148.164
C01379=1230.445,326.973,-69.776,-176.112,6.991,148.164
C01380=1230.441,327.222,-69.808,-176.110,6.994,148.164
C01381=1230.437,327.469,-69.838,-176.107,6.997,148.164
C01382=1230.433,327.717,-69.868,-176.106,6.999,148.164
C01383=1230.429,327.966,-69.900,-176.103,7.002,148.164
C01384=1230.424,328.214,-69.930,-176.102,7.005,148.164
C01385=1230.420,328.462,-69.961,-176.099,7.007,148.164
C01386=1230.416,328.710,-69.993,-176.097,7.009,148.164
C01387=1230.412,328.957,-70.023,-176.095,7.013,148.164
C01388=1230.407,329.205,-70.054,-176.093,7.015,148.164
C01389=1230.403,329.454,-70.085,-176.091,7.017,148.165
C01390=1230.399,329.702,-70.116,-176.089,7.020,148.165
C01391=1230.394,329.950,-70.147,-176.087,7.023,148.165
C01392=1230.390,330.198,-70.178,-176.085,7.025,148.165
C01393=1230.387,330.446,-70.209,-176.083,7.027,148.165
C01394=1230.382,330.694,-70.239,-176.081,7.031,148.165
C01395=1230.378,330.942,-70.270,-176.079,7.033,148.165
C01396=1230.373,331.190,-70.301,-176.077,7.035,148.165
C01397=1230.369,331.437,-70.333,-176.075,7.038,148.165
C01398=1230.365,331.686,-70.364,-176.073,7.041,148.165
C01399=1230.360,331.934,-70.395,-176.071,7.043,148.165
C01400=1230.356,332.183,-70.426,-176.069,7.046,148.165
C01401=1230.352,332.430,-70.457,-176.066,7.049,148.165
C01402=1230.347,332.678,-70.488,-176.065,7.051,148.166
C01403=1230.344,332.926,-70.518,-176.063,7.054,148.166
C01404=1230.340,333.174,-70.550,-176.061,7.056,148.166
C01405=1230.336,333.422,-70.581,-176.058,7.059,148.166
C01406=1230.331,333.670,-70.612,-176.057,7.062,148.166
C01407=1230.327,333.918,-70.643,-176.055,7.064,148.166
C01408=1230.323,334.166,-70.674,-176.053,7.067,148.166
C01409=1230.318,334.414,-70.705,-176.051,7.070,148.166
C01410=1230.315,334.662,-70.737,-176.049,7.072,148.166
C01411=1230.310,334.910,-70.768,-176.047,7.075,148.166
C01412=1230.306,335.159,-70.799,-176.045,7.078,148.166
C01413=1230.302,335.406,-70.830,-176.043,7.080,148.167
C01414=1230.297,335.654,-70.861,-176.041,7.083,148.167
C01415=1230.293,335.902,-70.893,-176.039,7.085,148.167
C01416=1230.289,336.150,-70.924,-176.037,7.088,148.167
C01417=1230.285,336.398,-70.956,-176.035,7.091,148.167
C01418=1230.280,336.646,-70.986,-176.033,7.093,148.167
C01419=1230.277,336.894,-71.018,-176.032,7.096,148.167
C01420=1230.272,337.142,-71.049,-176.029,7.099,148.167
C01421=1230.268,337.390,-71.081,-176.027,7.101,148.167
C01422=1230.264,337.638,-71.112,-176.025,7.104,148.167
C01423=1230.259,337.887,-71.144,-176.024,7.106,148.168
C01424=1230.255,338.135,-71.175,-176.022,7.109,148.168
C01425=1230.251,338.383,-71.207,-176.019,7.112,148.168
C01426=1230.246,338.631,-71.237,-176.018,7.114,148.168
C01427=1230.243,338.879,-71.269,-176.016,7.118,148.168
C01428=1230.238,339.127,-71.300,-176.014,7.120,148.168
C01429=1230.234,339.375,-71.332,-176.012,7.122,148.168
C01430=1230.230,339.622,-71.363,-176.010,7.125,148.169
C01431=1230.226,339.871,-71.395,-176.008,7.128,148.169
C01432=1230.222,340.118,-71.426,-176.006,7.130,148.169
C01433=1230.217,340.367,-71.458,-176.004,7.133,148.169
C01434=1230.213,340.614,-71.489,-176.003,7.136,148.169
C01435=1230.209,340.862,-71.521,-176.000,7.139,148.169
C01436=1230.204,341.140,-71.556,-175.999,7.141,148.169
C01437=1230.199,341.417,-71.591,-175.996,7.144,148.170
C01438=1230.195,341.695,-71.627,-175.994,7.147,148.170
C01439=1230.190,341.972,-71.661,-175.992,7.150,148.170
C01440=1230.185,342.221,-71.694,-175.990,7.153,148.170
C01441=1230.181,342.468,-71.725,-175.988,7.156,148.170
C01442=1230.177,342.717,-71.756,-175.986,7.158,148.170
C01443=1230.173,342.965,-71.788,-175.985,7.161,148.170
C01444=1230.169,343.212,-71.820,-175.983,7.163,148.170
C01445=1230.165,343.460,-71.852,-175.981,7.167,148.171
C01446=1230.160,343.708,-71.883,-175.979,7.169,148.171
C01447=1230.156,343.956,-71.915,-175.977,7.171,148.171
C01448=1230.152,344.204,-71.946,-175.975,7.174,148.171
C01449=1230.148,344.452,-71.979,-175.974,7.176,148.171
C01450=1230.144,344.700,-72.011,-175.972,7.180,148.171
C01451=1230.139,344.948,-72.041,-175.970,7.182,148.172
C01452=1230.136,345.196,-72.073,-175.968,7.185,148.172
C01453=1230.131,345.444,-72.105,-175.966,7.187,148.172
C01454=1230.127,345.692,-72.137,-175.964,7.191,148.172
C01455=1230.123,345.940,-72.169,-175.963,7.193,148.172
C01456=1230.118,346.187,-72.201,-175.961,7.196,148.172
C01457=1230.114,346.436,-72.232,-175.959,7.198,148.173
C01458=1230.110,346.683,-72.264,-175.958,7.201,148.173
C01459=1230.106,346.931,-72.295,-175.955,7.204,148.173
C01460=1230.102,347.180,-72.328,-175.954,7.207,148.173
C01461=1230.097,347.427,-72.359,-175.952,7.209,148.173
C01462=1230.094,347.675,-72.391,-175.950,7.211,148.173
C01463=1230.089,347.924,-72.424,-175.948,7.215,148.174
C01464=1230.085,348.171,-72.455,-175.946,7.217,148.174
C01465=1230.080,348.419,-72.488,-175.945,7.220,148.174
C01466=1230.076,348.667,-72.519,-175.943,7.222,148.174
C01467=1230.072,348.915,-72.551,-175.941,7.225,148.174
C01468=1230.068,349.163,-72.583,-175.939,7.228,148.175
C01469=1230.064,349.410,-72.615,-175.938,7.231,148.175
C01470=1230.060,349.658,-72.647,-175.936,7.233,148.175
C01471=1230.055,349.907,-72.679,-175.934,7.236,148.175
C01472=1230.051,350.154,-72.711,-175.933,7.238,148.175
C01473=1230.047,350.402,-72.743,-175.931,7.242,148.175
C01474=1230.043,350.650,-72.775,-175.929,7.244,148.176
C01475=1230.039,350.898,-72.806,-175.927,7.247,148.176
C01476=1230.034,351.146,-72.839,-175.926,7.249,148.176
C01477=1230.031,351.394,-72.871,-175.924,7.252,148.176
C01478=1230.026,351.642,-72.903,-175.922,7.255,148.176
C01479=1230.022,351.890,-72.935,-175.920,7.258,148.177
C01480=1230.018,352.138,-72.968,-175.919,7.260,148.177
C01481=1230.014,352.386,-73.000,-175.917,7.263,148.177
C01482=1230.009,352.633,-73.032,-175.915,7.265,148.177
C01483=1230.005,352.881,-73.063,-175.914,7.268,148.177
C01484=1230.001,353.130,-73.096,-175.912,7.271,148.178
C01485=1229.997,353.378,-73.128,-175.910,7.274,148.178
C01486=1229.992,353.625,-73.161,-175.908,7.276,148.178
C01487=1229.989,353.873,-73.192,-175.907,7.279,148.178
C01488=1229.984,354.121,-73.225,-175.906,7.282,148.179
C01489=1229.980,354.368,-73.256,-175.903,7.285,148.179
C01490=1229.975,354.617,-73.289,-175.902,7.287,148.179
C01491=1229.972,354.864,-73.321,-175.900,7.290,148.179
C01492=1229.968,355.113,-73.354,-175.899,7.293,148.179
C01493=1229.963,355.360,-73.385,-175.897,7.295,148.180
C01494=1229.959,355.608,-73.418,-175.895,7.298,148.180
C01495=1229.955,355.856,-73.450,-175.894,7.301,148.180
C01496=1229.951,356.104,-73.483,-175.892,7.304,148.180
C01497=1229.947,356.352,-73.514,-175.890,7.306,148.181
C01498=1229.942,356.600,-73.547,-175.889,7.309,148.181
C01499=1229.939,356.847,-73.579,-175.887,7.311,148.181
C01500=1229.934,357.095,-73.612,-175.886,7.314,148.181
C01501=1229.930,357.344,-73.644,-175.884,7.317,148.181
C01502=1229.926,357.590,-73.676,-175.882,7.320,148.182
C01503=1229.921,357.839,-73.709,-175.881,7.323,148.182
C01504=1229.918,358.087,-73.740,-175.879,7.325,148.182
C01505=1229.914,358.335,-73.774,-175.878,7.328,148.182
C01506=1229.909,358.583,-73.806,-175.876,7.331,148.183
C01507=1229.905,358.830,-73.838,-175.875,7.333,148.183
C01508=1229.901,359.078,-73.871,-175.873,7.336,148.183
C01509=1229.896,359.326,-73.903,-175.872,7.338,148.183
C01510=1229.893,359.574,-73.936,-175.870,7.342,148.184
C01511=1229.888,359.822,-73.968,-175.868,7.344,148.184
C01512=1229.885,360.070,-74.001,-175.866,7.347,148.184
C01513=1229.880,360.317,-74.033,-175.865,7.350,148.184
C01514=1229.876,360.565,-74.066,-175.864,7.352,148.185
C01515=1229.872,360.813,-74.098,-175.862,7.355,148.185
C01516=1229.868,361.061,-74.131,-175.861,7.358,148.185
C01517=1229.864,361.309,-74.163,-175.859,7.360,148.185
C01518=1229.860,361.556,-74.196,-175.858,7.363,148.186
C01519=1229.855,361.804,-74.228,-175.856,7.366,148.186
C01520=1229.851,362.052,-74.261,-175.854,7.369,148.186
C01521=1229.847,362.300,-74.294,-175.853,7.371,148.186
C01522=1229.843,362.548,-74.326,-175.851,7.374,148.187
C01523=1229.839,362.796,-74.359,-175.850,7.377,148.187
C01524=1229.835,363.044,-74.392,-175.848,7.379,148.187
C01525=1229.831,363.292,-74.424,-175.847,7.382,148.188
C01526=1229.826,363.539,-74.456,-175.845,7.385,148.188
C01527=1229.822,363.787,-74.489,-175.844,7.387,148.188
C01528=1229.818,364.035,-74.522,-175.843,7.390,148.188
C01529=1229.814,364.282,-74.555,-175.841,7.392,148.189
C01530=1229.810,364.531,-74.587,-175.840,7.395,148.189
C01531=1229.806,364.778,-74.620,-175.838,7.398,148.189
C01532=1229.801,365.027,-74.653,-175.836,7.402,148.190
C01533=1229.798,365.274,-74.685,-175.835,7.404,148.190
C01534=1229.794,365.522,-74.718,-175.834,7.407,148.190
C01535=1229.789,365.770,-74.751,-175.832,7.409,148.190
C01536=1229.784,366.017,-74.784,-175.831,7.412,148.191
C01537=1229.780,366.265,-74.817,-175.829,7.415,148.191
C01538=1229.777,366.513,-74.849,-175.828,7.418,148.191
C01539=1229.772,366.761,-74.882,-175.826,7.420,148.192
C01540=1229.768,367.040,-74.919,-175.825,7.423,148.192
C01541=1229.763,367.320,-74.956,-175.823,7.426,148.192
C01542=1229.758,367.599,-74.993,-175.822,7.429,148.193
C01543=1229.754,367.879,-75.030,-175.821,7.432,148.193
C01544=1229.750,368.126,-75.063,-175.819,7.434,148.193
C01545=1229.745,368.375,-75.096,-175.818,7.437,148.194
C01546=1229.741,368.622,-75.129,-175.816,7.440,148.194
C01547=1229.737,368.870,-75.162,-175.815,7.443,148.194
C01548=1229.734,369.118,-75.195,-175.814,7.445,148.194
C01549=1229.729,369.366,-75.227,-175.812,7.448,148.195
C01550=1229.725,369.614,-75.260,-175.811,7.451,148.195
C01551=1229.721,369.861,-75.293,-175.810,7.453,148.195
C01552=1229.717,370.109,-75.327,-175.808,7.456,148.196
C01553=1229.713,370.357,-75.360,-175.807,7.459,148.196
C01554=1229.708,370.605,-75.392,-175.806,7.462,148.196
C01555=1229.704,370.853,-75.425,-175.805,7.464,148.197
C01556=1229.700,371.101,-75.458,-175.803,7.467,148.197
C01557=1229.696,371.348,-75.492,-175.802,7.470,148.197
C01558=1229.692,371.596,-75.525,-175.801,7.473,148.198
C01559=1229.688,371.844,-75.557,-175.799,7.475,148.198
C01560=1229.684,372.091,-75.590,-175.798,7.478,148.198
C01561=1229.680,372.339,-75.624,-175.797,7.481,148.199
C01562=1229.675,372.587,-75.656,-175.795,7.483,148.199
C01563=1229.671,372.835,-75.689,-175.794,7.486,148.199
C01564=1229.667,373.083,-75.722,-175.793,7.489,148.200
C01565=1229.663,373.331,-75.756,-175.791,7.491,148.200
C01566=1229.659,373.578,-75.789,-175.790,7.493,148.200
C01567=1229.655,373.826,-75.822,-175.789,7.496,148.201
C01568=1229.651,374.074,-75.855,-175.788,7.499,148.201
C01569=1229.647,374.321,-75.888,-175.786,7.502,148.201
C01570=1229.642,374.569,-75.921,-175.785,7.504,148.202
C01571=1229.638,374.817,-75.954,-175.784,7.507,148.202
C01572=1229.634,375.065,-75.988,-175.783,7.510,148.202
C01573=1229.630,375.312,-76.021,-175.781,7.513,148.203
C01574=1229.626,375.560,-76.054,-175.780,7.515,148.203
C01575=1229.622,375.808,-76.087,-175.780,7.517,148.203
C01576=1229.618,376.056,-76.120,-175.778,7.520,148.204
C01577=1229.613,376.303,-76.153,-175.777,7.523,148.204
C01578=1229.609,376.551,-76.187,-175.776,7.526,148.204
C01579=1229.605,376.799,-76.220,-175.774,7.528,148.205
C01580=1229.601,377.046,-76.253,-175.773,7.531,148.205
C01581=1229.597,377.294,-76.286,-175.773,7.533,148.205
C01582=1229.593,377.542,-76.319,-175.772,7.536,148.206
C01583=1229.588,377.789,-76.354,-175.770,7.539,148.206
C01584=1229.584,378.037,-76.387,-175.769,7.541,148.206
C01585=1229.580,378.285,-76.420,-175.768,7.544,148.207
C01586=1229.576,378.533,-76.453,-175.766,7.547,148.207
C01587=1229.572,378.781,-76.487,-175.766,7.549,148.208
C01588=1229.568,379.029,-76.520,-175.765,7.552,148.208
C01589=1229.564,379.276,-76.553,-175.763,7.555,148.208
C01590=1229.560,379.524,-76.586,-175.762,7.557,148.209
C01591=1229.556,379.772,-76.619,-175.761,7.560,148.209
C01592=1229.552,380.019,-76.653,-175.760,7.562,148.209
C01593=1229.547,380.267,-76.687,-175.759,7.565,148.210
C01594=1229.543,380.515,-76.720,-175.758,7.568,148.210
C01595=1229.539,380.762,-76.753,-175.757,7.571,148.211
C01596=1229.535,381.010,-76.786,-175.756,7.573,148.211
C01597=1229.531,381.258,-76.821,-175.755,7.575,148.211
C01598=1229.527,381.506,-76.854,-175.754,7.578,148.212
C01599=1229.523,381.753,-76.887,-175.752,7.581,148.212
C01600=1229.518,382.002,-76.921,-175.752,7.583,148.212
C01601=1229.514,382.249,-76.954,-175.751,7.586,148.213
C01602=1229.510,382.496,-76.988,-175.749,7.588,148.213
C01603=1229.506,382.744,-77.021,-175.748,7.591,148.213
C01604=1229.502,382.992,-77.054,-175.747,7.593,148.214
C01605=1229.498,383.240,-77.087,-175.746,7.596,148.214
C01606=1229.494,383.488,-77.122,-175.745,7.599,148.215
C01607=1229.490,383.735,-77.155,-175.744,7.601,148.215
C01608=1229.486,383.983,-77.188,-175.743,7.604,148.215
C01609=1229.482,384.230,-77.222,-175.742,7.606,148.216
C01610=1229.478,384.478,-77.255,-175.741,7.609,148.216
C01611=1229.473,384.726,-77.289,-175.740,7.611,148.216
C01612=1229.469,384.973,-77.323,-175.739,7.614,148.217
C01613=1229.465,385.222,-77.356,-175.738,7.617,148.217
C01614=1229.461,385.469,-77.390,-175.737,7.619,148.218
C01615=1229.457,385.716,-77.423,-175.736,7.622,148.218
C01616=1229.452,385.964,-77.457,-175.735,7.624,148.218
C01617=1229.448,386.212,-77.490,-175.734,7.626,148.219
C01618=1229.444,386.459,-77.524,-175.733,7.629,148.219
C01619=1229.441,386.708,-77.558,-175.732,7.632,148.220
C01620=1229.436,386.956,-77.592,-175.732,7.634,148.220
C01621=1229.432,387.203,-77.625,-175.731,7.637,148.220
C01622=1229.428,387.451,-77.659,-175.729,7.640,148.221
C01623=1229.424,387.698,-77.692,-175.729,7.642,148.221
C01624=1229.419,387.946,-77.726,-175.728,7.645,148.222
C01625=1229.416,388.194,-77.760,-175.727,7.647,148.222
C01626=1229.412,388.441,-77.794,-175.726,7.650,148.222
C01627=1229.407,388.689,-77.827,-175.725,7.652,148.223
C01628=1229.403,388.936,-77.861,-175.724,7.654,148.223
C01629=1229.399,389.184,-77.894,-175.723,7.657,148.223
C01630=1229.396,389.432,-77.929,-175.722,7.659,148.224
C01631=1229.391,389.680,-77.962,-175.721,7.662,148.224
C01632=1229.387,389.927,-77.996,-175.720,7.665,148.225
C01633=1229.383,390.175,-78.029,-175.720,7.667,148.225
C01634=1229.378,390.423,-78.063,-175.719,7.670,148.226
C01635=1229.375,390.671,-78.097,-175.718,7.672,148.226
C01636=1229.371,390.918,-78.131,-175.717,7.675,148.226
C01637=1229.366,391.166,-78.165,-175.716,7.677,148.227
C01638=1229.362,391.414,-78.198,-175.715,7.680,148.227
C01639=1229.359,391.661,-78.232,-175.714,7.682,148.227
C01640=1229.354,391.909,-78.267,-175.713,7.684,148.228
C01641=1229.350,392.157,-78.300,-175.712,7.688,148.228
C01642=1229.346,392.404,-78.334,-175.712,7.690,148.229
C01643=1229.342,392.652,-78.368,-175.711,7.692,148.229
C01644=1229.337,392.933,-78.406,-175.709,7.695,148.230
C01645=1229.333,393.215,-78.445,-175.709,7.697,148.230
C01646=1229.328,393.496,-78.483,-175.708,7.700,148.230
C01647=1229.324,393.777,-78.521,-175.707,7.703,148.231
C01648=1229.319,394.025,-78.556,-175.706,7.706,148.231
C01649=1229.315,394.272,-78.590,-175.706,7.708,148.232
C01650=1229.311,394.521,-78.624,-175.704,7.711,148.232
C01651=1229.307,394.768,-78.658,-175.704,7.713,148.233
C01652=1229.303,395.016,-78.691,-175.703,7.716,148.233
C01653=1229.299,395.263,-78.725,-175.702,7.718,148.233
C01654=1229.295,395.511,-78.759,-175.701,7.721,148.234
C01655=1229.290,395.759,-78.793,-175.701,7.723,148.234
C01656=1229.287,396.006,-78.827,-175.700,7.725,148.235
C01657=1229.283,396.254,-78.861,-175.699,7.728,148.235
C01658=1229.278,396.502,-78.895,-175.698,7.730,148.235
C01659=1229.275,396.749,-78.929,-175.697,7.732,148.236
C01660=1229.270,396.996,-78.963,-175.697,7.735,148.236
C01661=1229.267,397.245,-78.997,-175.696,7.738,148.237
C01662=1229.262,397.492,-79.031,-175.695,7.740,148.237
C01663=1229.258,397.739,-79.065,-175.694,7.742,148.237
C01664=1229.254,397.988,-79.099,-175.693,7.744,148.238
C01665=1229.250,398.235,-79.133,-175.693,7.747,148.238
C01666=1229.245,398.483,-79.168,-175.692,7.749,148.239
C01667=1229.241,398.730,-79.201,-175.691,7.751,148.239
C01668=1229.238,398.978,-79.235,-175.690,7.754,148.239
C01669=1229.234,399.226,-79.270,-175.690,7.757,148.240
C01670=1229.230,399.473,-79.303,-175.689,7.759,148.240
C01671=1229.225,399.721,-79.338,-175.688,7.761,148.241
C01672=1229.222,399.969,-79.371,-175.688,7.763,148.241
C01673=1229.217,400.216,-79.406,-175.686,7.766,148.242
C01674=1229.214,400.464,-79.440,-175.686,7.768,148.242
C01675=1229.209,400.712,-79.474,-175.686,7.770,148.242
C01676=1229.205,400.959,-79.508,-175.684,7.773,148.243
C01677=1229.201,401.206,-79.542,-175.684,7.775,148.243
C01678=1229.197,401.454,-79.576,-175.684,7.777,148.244
C01679=1229.193,401.702,-79.611,-175.682,7.780,148.244
C01680=1229.189,401.949,-79.644,-175.682,7.782,148.244
C01681=1229.185,402.197,-79.679,-175.681,7.784,148.245
C01682=1229.180,402.445,-79.713,-175.681,7.787,148.245
C01683=1229.176,402.692,-79.747,-175.680,7.789,148.246
C01684=1229.172,402.940,-79.782,-175.679,7.791,148.246
C01685=1229.168,403.187,-79.816,-175.678,7.794,148.246
C01686=1229.164,403.435,-79.850,-175.678,7.796,148.247
C01687=1229.160,403.683,-79.884,-175.677,7.798,148.247
C01688=1229.156,403.930,-79.918,-175.676,7.801,148.248
C01689=1229.152,404.178,-79.953,-175.675,7.803,148.248
C01690=1229.148,404.426,-79.987,-175.675,7.805,148.249
C01691=1229.144,404.673,-80.021,-175.674,7.808,148.249
C01692=1229.140,404.921,-80.056,-175.673,7.810,148.249
C01693=1229.136,405.168,-80.090,-175.673,7.812,148.250
C01694=1229.131,405.416,-80.123,-175.673,7.815,148.250
C01695=1229.127,405.664,-80.158,-175.672,7.817,148.251
C01696=1229.124,405.911,-80.192,-175.671,7.819,148.251
C01697=1229.119,406.159,-80.227,-175.671,7.822,148.252
C01698=1229.115,406.407,-80.261,-175.670,7.824,148.252
C01699=1229.111,406.654,-80.295,-175.669,7.826,148.252
C01700=1229.107,406.902,-80.330,-175.668,7.828,148.253
C01701=1229.103,407.149,-80.364,-175.668,7.831,148.253
C01702=1229.099,407.397,-80.398,-175.667,7.833,148.254
C01703=1229.095,407.645,-80.433,-175.666,7.835,148.254
C01704=1229.091,407.892,-80.467,-175.666,7.837,148.254
C01705=1229.087,408.139,-80.502,-175.665,7.840,148.255
C01706=1229.083,408.387,-80.536,-175.665,7.842,148.255
C01707=1229.079,408.634,-80.570,-175.664,7.845,148.256
C01708=1229.075,408.883,-80.605,-175.664,7.847,148.256
C01709=1229.071,409.130,-80.639,-175.663,7.849,148.256
C01710=1229.066,409.377,-80.674,-175.662,7.851,148.257
C01711=1229.062,409.625,-80.708,-175.661,7.854,148.257
C01712=1229.059,409.872,-80.742,-175.661,7.856,148.258
C01713=1229.055,410.120,-80.777,-175.660,7.858,148.258
C01714=1229.050,410.368,-80.812,-175.660,7.860,148.258
C01715=1229.047,410.616,-80.846,-175.659,7.862,148.259
C01716=1229.042,410.863,-80.880,-175.658,7.865,148.259
C01717=1229.038,411.110,-80.915,-175.658,7.867,148.260
C01718=1229.034,411.358,-80.949,-175.657,7.869,148.260
C01719=1229.030,411.606,-80.983,-175.657,7.871,148.261
C01720=1229.026,411.854,-81.018,-175.656,7.873,148.261
C01721=1229.022,412.101,-81.052,-175.656,7.875,148.261
C01722=1229.017,412.348,-81.087,-175.654,7.878,148.262
C01723=1229.013,412.596,-81.121,-175.654,7.880,148.262
C01724=1229.010,412.844,-81.155,-175.654,7.882,148.263
C01725=1229.006,413.092,-81.190,-175.653,7.884,148.263
C01726=1229.001,413.339,-81.225,-175.652,7.886,148.263
C01727=1228.998,413.587,-81.259,-175.652,7.888,148.264
C01728=1228.994,413.834,-81.294,-175.651,7.891,148.264
C01729=1228.989,414.081,-81.328,-175.650,7.893,148.265
C01730=1228.986,414.329,-81.363,-175.650,7.895,148.265
C01731=1228.981,414.576,-81.397,-175.650,7.897,148.265
C01732=1228.977,414.825,-81.432,-175.649,7.899,148.266
C01733=1228.973,415.072,-81.466,-175.648,7.901,148.266
C01734=1228.969,415.320,-81.501,-175.648,7.904,148.267
C01735=1228.965,415.567,-81.535,-175.647,7.906,148.267
C01736=1228.959,415.949,-81.589,-175.646,7.910,148.268
C01737=1228.952,416.330,-81.642,-175.645,7.913,148.268
C01738=1228.946,416.713,-81.695,-175.645,7.916,148.269
C01739=1228.942,417.095,-81.749,-175.644,7.919,148.269
C01740=1228.519,417.094,-81.781,-175.647,7.929,148.273
C01741=1228.524,416.710,-81.728,-175.648,7.926,148.272
C01742=1228.530,416.325,-81.674,-175.649,7.923,148.272
C01743=1228.537,415.941,-81.621,-175.649,7.920,148.271
C01744=1228.543,415.556,-81.567,-175.651,7.916,148.271
C01745=1228.547,415.309,-81.532,-175.651,7.914,148.270
C01746=1228.551,415.061,-81.497,-175.652,7.912,148.270
C01747=1228.555,414.814,-81.463,-175.652,7.910,148.269
C01748=1228.560,414.567,-81.428,-175.653,7.908,148.269
C01749=1228.563,414.319,-81.394,-175.653,7.906,148.269
C01750=1228.568,414.071,-81.360,-175.654,7.904,148.268
C01751=1228.572,413.823,-81.325,-175.655,7.901,148.268
C01752=1228.575,413.576,-81.291,-175.655,7.899,148.267
C01753=1228.579,413.329,-81.256,-175.656,7.897,148.267
C01754=1228.584,413.081,-81.221,-175.656,7.895,148.267
C01755=1228.588,412.833,-81.186,-175.657,7.892,148.266
C01756=1228.592,412.586,-81.152,-175.657,7.891,148.266
C01757=1228.596,412.338,-81.118,-175.658,7.889,148.265
C01758=1228.600,412.090,-81.083,-175.659,7.885,148.265
C01759=1228.604,411.843,-81.049,-175.659,7.883,148.265
C01760=1228.608,411.595,-81.014,-175.660,7.881,148.264
C01761=1228.612,411.348,-80.980,-175.661,7.879,148.264
C01762=1228.616,411.100,-80.946,-175.661,7.877,148.263
C01763=1228.620,410.852,-80.911,-175.662,7.874,148.263
C01764=1228.625,410.605,-80.877,-175.663,7.872,148.263
C01765=1228.628,410.357,-80.842,-175.663,7.870,148.262
C01766=1228.633,410.110,-80.808,-175.663,7.868,148.262
C01767=1228.637,409.862,-80.773,-175.664,7.866,148.261
C01768=1228.640,409.615,-80.739,-175.665,7.863,148.261
C01769=1228.645,409.367,-80.705,-175.665,7.861,148.260
C01770=1228.649,409.119,-80.670,-175.666,7.859,148.260
C01771=1228.653,408.872,-80.636,-175.667,7.857,148.260
C01772=1228.657,408.624,-80.601,-175.667,7.855,148.259
C01773=1228.661,408.377,-80.567,-175.668,7.852,148.259
C01774=1228.665,408.129,-80.533,-175.669,7.850,148.258
C01775=1228.669,407.881,-80.498,-175.669,7.848,148.258
C01776=1228.673,407.634,-80.464,-175.669,7.846,148.258
C01777=1228.677,407.386,-80.429,-175.671,7.843,148.257
C01778=1228.681,407.139,-80.395,-175.671,7.841,148.257
C01779=1228.685,406.891,-80.361,-175.672,7.839,148.256
C01780=1228.689,406.643,-80.326,-175.672,7.837,148.256
C01781=1228.693,406.396,-80.292,-175.673,7.834,148.255
C01782=1228.698,406.149,-80.258,-175.674,7.832,148.255
C01783=1228.702,405.901,-80.223,-175.674,7.830,148.255
C01784=1228.705,405.654,-80.189,-175.675,7.828,148.254
C01785=1228.709,405.405,-80.154,-175.676,7.825,148.254
C01786=1228.713,405.158,-80.121,-175.676,7.823,148.254
C01787=1228.718,404.911,-80.086,-175.677,7.821,148.253
C01788=1228.721,404.662,-80.053,-175.677,7.819,148.253
C01789=1228.726,404.415,-80.018,-175.678,7.816,148.252
C01790=1228.731,404.168,-79.984,-175.679,7.814,148.252
C01791=1228.734,403.920,-79.949,-175.679,7.812,148.251
C01792=1228.738,403.672,-79.915,-175.680,7.809,148.251
C01793=1228.742,403.425,-79.881,-175.681,7.807,148.251
C01794=1228.746,403.177,-79.846,-175.681,7.804,148.250
C01795=1228.750,402.930,-79.812,-175.682,7.802,148.250
C01796=1228.754,402.681,-79.778,-175.683,7.800,148.249
C01797=1228.758,402.434,-79.744,-175.684,7.798,148.249
C01798=1228.763,402.187,-79.710,-175.684,7.795,148.248
C01799=1228.767,401.939,-79.675,-175.685,7.793,148.248
C01800=1228.770,401.692,-79.641,-175.686,7.791,148.248
C01801=1228.775,401.444,-79.607,-175.687,7.788,148.247
C01802=1228.779,401.196,-79.573,-175.687,7.786,148.247
C01803=1228.783,400.948,-79.539,-175.688,7.784,148.246
C01804=1228.787,400.701,-79.505,-175.689,7.781,148.246
C01805=1228.792,400.454,-79.470,-175.689,7.779,148.246
C01806=1228.795,400.205,-79.437,-175.690,7.776,148.245
C01807=1228.800,399.958,-79.402,-175.691,7.774,148.245
C01808=1228.803,399.711,-79.369,-175.691,7.772,148.244
C01809=1228.807,399.463,-79.334,-175.692,7.769,148.244
C01810=1228.812,399.215,-79.301,-175.693,7.767,148.243
C01811=1228.816,398.968,-79.266,-175.693,7.765,148.243
C01812=1228.819,398.720,-79.232,-175.694,7.762,148.243
C01813=1228.824,398.472,-79.197,-175.695,7.760,148.242
C01814=1228.828,398.225,-79.164,-175.696,7.757,148.242
C01815=1228.832,397.976,-79.129,-175.696,7.755,148.241
C01816=1228.836,397.729,-79.096,-175.697,7.753,148.241
C01817=1228.840,397.482,-79.062,-175.698,7.750,148.241
C01818=1228.845,397.234,-79.028,-175.699,7.748,148.240
